LIN {X 0,Y 580.933,Z 477.254,A -85,B 0,C 180,E1 -1786.489,E2 -1786.489} C_VEL
LIN {X 0,Y 580.805,Z 577.725,A -85,B 0,C 180,E1 -1787.752,E2 -1787.752} C_VEL
LIN {X 0,Y 580.706,Z 590.474,A -85,B 0,C 180,E1 -1788.038,E2 -1788.038} C_VEL
LIN {X 0,Y 580.629,Z 603.373,A -85,B 0,C 180,E1 -1788.48,E2 -1788.48} C_VEL
LIN {X 0,Y 580.569,Z 614.719,A -85,B 0,C 180,E1 -1789.009,E2 -1789.009} C_VEL
LIN {X 0,Y 580.47,Z 626.557,A -85,B 0,C 180,E1 -1789.713,E2 -1789.713} C_VEL
LIN {X 0,Y 580.367,Z 638.111,A -85,B 0,C 180,E1 -1790.591,E2 -1790.591} C_VEL
LIN {X 0,Y 580.281,Z 647.332,A -85,B 0,C 180,E1 -1791.468,E2 -1791.468} C_VEL
LIN {X 0,Y 580.221,Z 654.959,A -85,B 0,C 180,E1 -1792.343,E2 -1792.343} C_VEL
LIN {X 0,Y 580.171,Z 662.355,A -85,B 0,C 180,E1 -1793.377,E2 -1793.377} C_VEL
LIN {X 0,Y 580.138,Z 668.453,A -85,B 0,C 180,E1 -1794.438,E2 -1794.438} C_VEL
LIN {X 0,Y 580.107,Z 673.197,A -85,B 0,C 180,E1 -1795.483,E2 -1795.483} C_VEL
LIN {X 0,Y 580.123,Z 676.829,A -85,B 0,C 180,E1 -1796.527,E2 -1796.527} C_VEL
LIN {X 0,Y 580.043,Z 678.681,A -85,B 0,C 180,E1 -1797.222,E2 -1797.222} C_VEL
LIN {X 0,Y 580.046,Z 681.138,A -85,B 0,C 180,E1 -1798.611,E2 -1798.611} C_VEL
LIN {X 0,Y 580.041,Z 681.753,A -85,B 0,C 180,E1 -1799.306,E2 -1799.306} C_VEL
LIN {X 0,Y 580.04,Z 681.812,A -85,B 0,C 180,E1 -1800.694,E2 -1800.694} C_VEL
LIN {X 0,Y 580.047,Z 681.24,A -85,B 0,C 180,E1 -1801.389,E2 -1801.389} C_VEL
LIN {X 0,Y 580.044,Z 678.908,A -85,B 0,C 180,E1 -1802.778,E2 -1802.778} C_VEL
LIN {X 0,Y 580.11,Z 676.037,A -85,B 0,C 180,E1 -1803.821,E2 -1803.821} C_VEL
LIN {X 0,Y 580.053,Z 672.134,A -85,B 0,C 180,E1 -1804.865,E2 -1804.865} C_VEL
LIN {X 0,Y 580.162,Z 667.083,A -85,B 0,C 180,E1 -1805.91,E2 -1805.91} C_VEL
LIN {X 0,Y 580.157,Z 660.739,A -85,B 0,C 180,E1 -1806.958,E2 -1806.958} C_VEL
LIN {X 0,Y 580.241,Z 652.871,A -85,B 0,C 180,E1 -1808.007,E2 -1808.007} C_VEL
LIN {X 0,Y 580.308,Z 643.003,A -85,B 0,C 180,E1 -1809.058,E2 -1809.058} C_VEL
LIN {X 0,Y 580.392,Z 633.8,A -85,B 0,C 180,E1 -1809.848,E2 -1809.848} C_VEL
LIN {X 0,Y 580.498,Z 623.854,A -85,B 0,C 180,E1 -1810.551,E2 -1810.551} C_VEL
LIN {X 0,Y 580.609,Z 613.074,A -85,B 0,C 180,E1 -1811.167,E2 -1811.167} C_VEL
LIN {X 0,Y 580.642,Z 600.005,A -85,B 0,C 180,E1 -1811.741,E2 -1811.741} C_VEL
LIN {X 0,Y 580.739,Z 587.106,A -85,B 0,C 180,E1 -1812.138,E2 -1812.138} C_VEL
LIN {X 0,Y 580.789,Z 575.132,A -85,B 0,C 180,E1 -1812.381,E2 -1812.381} C_VEL
LIN {X 0,Y 580.811,Z 472.633,A -85,B 0,C 180,E1 -1813.662,E2 -1813.662} C_VEL
LIN {X 0,Y 580.398,Z 469.615,A -85,B 0,C 180,E1 -1813.725,E2 -1813.725} C_VEL
LIN {X 0,Y 580.566,Z 448.09,A -85,B 0,C 180,E1 -1816.709,E2 -1816.709} C_VEL
LIN {X 0,Y 580.771,Z 427.235,A -85,B 0,C 180,E1 -1819.641,E2 -1819.641} C_VEL
LIN {X 0,Y 580.959,Z 406.656,A -85,B 0,C 180,E1 -1822.587,E2 -1822.587} C_VEL
LIN {X 0,Y 580.331,Z 401.637,A -85,B 0,C 180,E1 -1823.343,E2 -1823.343} C_VEL
LIN {X 0,Y 580.262,Z 401.208,A -85,B 0,C 180,E1 -1823.417,E2 -1823.417} C_VEL
LIN {X 0,Y 580.26,Z 401.203,A -85,B 0,C 180,E1 -1826.327,E2 -1826.327} C_VEL
LIN {X 0,Y 580.278,Z 401.204,A -85,B 0,C 180,E1 -1829.305,E2 -1829.305} C_VEL
LIN {X 0,Y 580.296,Z 401.197,A -85,B 0,C 180,E1 -1832.201,E2 -1832.201} C_VEL
LIN {X 0,Y 580.288,Z 401.198,A -85,B 0,C 180,E1 -1834.697,E2 -1834.697} C_VEL
LIN {X 0,Y 580.291,Z 401.205,A -85,B 0,C 180,E1 -1837.269,E2 -1837.269} C_VEL
LIN {X 0,Y 580.293,Z 401.196,A -85,B 0,C 180,E1 -1840.27,E2 -1840.27} C_VEL
LIN {X 0,Y 580.28,Z 401.202,A -85,B 0,C 180,E1 -1842.706,E2 -1842.706} C_VEL
LIN {X 0,Y 580.274,Z 401.2,A -85,B 0,C 180,E1 -1845.609,E2 -1845.609} C_VEL
LIN {X 0,Y 580.284,Z 401.199,A -85,B 0,C 180,E1 -1848.231,E2 -1848.231} C_VEL
LIN {X 0,Y 580.277,Z 401.205,A -85,B 0,C 180,E1 -1850.965,E2 -1850.965} C_VEL
LIN {X 0,Y 580.251,Z 401.201,A -85,B 0,C 180,E1 -1853.595,E2 -1853.595} C_VEL
LIN {X 0,Y 580.315,Z 401.197,A -85,B 0,C 180,E1 -1856.145,E2 -1856.145} C_VEL
LIN {X 0,Y 580.269,Z 401.207,A -85,B 0,C 180,E1 -1858.614,E2 -1858.614} C_VEL
LIN {X 0,Y 580.285,Z 401.2,A -85,B 0,C 180,E1 -1861.023,E2 -1861.023} C_VEL
LIN {X 0,Y 580.301,Z 401.201,A -85,B 0,C 180,E1 -1864.344,E2 -1864.344} C_VEL
LIN {X 0,Y 581.342,Z 407.343,A -85,B 0,C 180,E1 -1865.202,E2 -1865.202} C_VEL
LIN {X 0,Y 581.077,Z 429.583,A -85,B 0,C 180,E1 -1867.979,E2 -1867.979} C_VEL
LIN {X 0,Y 580.889,Z 450.217,A -85,B 0,C 180,E1 -1870.512,E2 -1870.512} C_VEL
LIN {X 0,Y 580.646,Z 473.238,A -85,B 0,C 180,E1 -1873.294,E2 -1873.294} C_VEL
LIN {X 0,Y 580.433,Z 498.075,A -85,B 0,C 180,E1 -1876.254,E2 -1876.254} C_VEL
LIN {X 0,Y 580.423,Z 498.64,A -85,B 0,C 180,E1 -1876.32,E2 -1876.32} C_VEL
LIN {X 0,Y 580.919,Z 503.714,A -85,B 0,C 180,E1 -1876.399,E2 -1876.399} C_VEL
LIN {X 0,Y 580.797,Z 607.943,A -85,B 0,C 180,E1 -1877.708,E2 -1877.708} C_VEL
LIN {X 0,Y 580.735,Z 621.217,A -85,B 0,C 180,E1 -1878.017,E2 -1878.017} C_VEL
LIN {X 0,Y 580.644,Z 634.148,A -85,B 0,C 180,E1 -1878.467,E2 -1878.467} C_VEL
LIN {X 0,Y 580.556,Z 645.629,A -85,B 0,C 180,E1 -1879.008,E2 -1879.008} C_VEL
LIN {X 0,Y 580.428,Z 657.202,A -85,B 0,C 180,E1 -1879.712,E2 -1879.712} C_VEL
LIN {X 0,Y 580.344,Z 667.598,A -85,B 0,C 180,E1 -1880.503,E2 -1880.503} C_VEL
LIN {X 0,Y 580.271,Z 676.112,A -85,B 0,C 180,E1 -1881.292,E2 -1881.292} C_VEL
LIN {X 0,Y 580.222,Z 683.96,A -85,B 0,C 180,E1 -1882.168,E2 -1882.168} C_VEL
LIN {X 0,Y 580.154,Z 691.65,A -85,B 0,C 180,E1 -1883.222,E2 -1883.222} C_VEL
LIN {X 0,Y 580.139,Z 698.68,A -85,B 0,C 180,E1 -1884.438,E2 -1884.438} C_VEL
LIN {X 0,Y 580.108,Z 703.372,A -85,B 0,C 180,E1 -1885.483,E2 -1885.483} C_VEL
LIN {X 0,Y 580.123,Z 706.957,A -85,B 0,C 180,E1 -1886.527,E2 -1886.527} C_VEL
LIN {X 0,Y 580.043,Z 708.808,A -85,B 0,C 180,E1 -1887.222,E2 -1887.222} C_VEL
LIN {X 0,Y 580.039,Z 710.199,A -85,B 0,C 180,E1 -1887.917,E2 -1887.917} C_VEL
LIN {X 0,Y 580.04,Z 711.785,A -85,B 0,C 180,E1 -1889.306,E2 -1889.306} C_VEL
LIN {X 0,Y 580.037,Z 712,A -85,B 0,C 180,E1 -1890,E2 -1890} C_VEL
LIN {X 0,Y 580.046,Z 711.186,A -85,B 0,C 180,E1 -1891.389,E2 -1891.389} C_VEL
LIN {X 0,Y 580.039,Z 710.2,A -85,B 0,C 180,E1 -1892.083,E2 -1892.083} C_VEL
LIN {X 0,Y 580.043,Z 708.81,A -85,B 0,C 180,E1 -1892.778,E2 -1892.778} C_VEL
LIN {X 0,Y 580.11,Z 705.896,A -85,B 0,C 180,E1 -1893.821,E2 -1893.821} C_VEL
LIN {X 0,Y 580.053,Z 701.949,A -85,B 0,C 180,E1 -1894.865,E2 -1894.865} C_VEL
LIN {X 0,Y 580.139,Z 695.877,A -85,B 0,C 180,E1 -1896.085,E2 -1896.085} C_VEL
LIN {X 0,Y 580.184,Z 689.237,A -85,B 0,C 180,E1 -1897.132,E2 -1897.132} C_VEL
LIN {X 0,Y 580.251,Z 680.99,A -85,B 0,C 180,E1 -1898.182,E2 -1898.182} C_VEL
LIN {X 0,Y 580.308,Z 672.537,A -85,B 0,C 180,E1 -1899.058,E2 -1899.058} C_VEL
LIN {X 0,Y 580.419,Z 662.096,A -85,B 0,C 180,E1 -1899.936,E2 -1899.936} C_VEL
LIN {X 0,Y 580.512,Z 651.756,A -85,B 0,C 180,E1 -1900.639,E2 -1900.639} C_VEL
LIN {X 0,Y 580.581,Z 640.408,A -85,B 0,C 180,E1 -1901.256,E2 -1901.256} C_VEL
LIN {X 0,Y 580.65,Z 628.765,A -85,B 0,C 180,E1 -1901.741,E2 -1901.741} C_VEL
LIN {X 0,Y 580.748,Z 615.347,A -85,B 0,C 180,E1 -1902.138,E2 -1902.138} C_VEL
LIN {X 0,Y 580.817,Z 602.079,A -85,B 0,C 180,E1 -1902.38,E2 -1902.38} C_VEL
LIN {X 0,Y 580.879,Z 501.925,A -85,B 0,C 180,E1 -1903.624,E2 -1903.624} C_VEL
LIN {X 0,Y 580.424,Z 498.452,A -85,B 0,C 180,E1 -1903.702,E2 -1903.702} C_VEL
LIN {X 0,Y 580.636,Z 474.743,A -85,B 0,C 180,E1 -1906.526,E2 -1906.526} C_VEL
LIN {X 0,Y 580.87,Z 451.661,A -85,B 0,C 180,E1 -1909.312,E2 -1909.312} C_VEL
LIN {X 0,Y 581.077,Z 429.583,A -85,B 0,C 180,E1 -1912.021,E2 -1912.021} C_VEL
LIN {X 0,Y 581.331,Z 407.325,A -85,B 0,C 180,E1 -1914.801,E2 -1914.801} C_VEL
LIN {X 0,Y 580.288,Z 401.206,A -85,B 0,C 180,E1 -1915.633,E2 -1915.633} C_VEL
LIN {X 0,Y 580.248,Z 401.205,A -85,B 0,C 180,E1 -1918.188,E2 -1918.188} C_VEL
LIN {X 0,Y 580.271,Z 401.2,A -85,B 0,C 180,E1 -1920.692,E2 -1920.692} C_VEL
LIN {X 0,Y 580.304,Z 401.201,A -85,B 0,C 180,E1 -1923.316,E2 -1923.316} C_VEL
LIN {X 0,Y 580.234,Z 401.209,A -85,B 0,C 180,E1 -1925.754,E2 -1925.754} C_VEL
LIN {X 0,Y 580.286,Z 401.198,A -85,B 0,C 180,E1 -1928.147,E2 -1928.147} C_VEL
LIN {X 0,Y 580.298,Z 401.198,A -85,B 0,C 180,E1 -1930.844,E2 -1930.844} C_VEL
LIN {X 0,Y 580.273,Z 401.203,A -85,B 0,C 180,E1 -1933.659,E2 -1933.659} C_VEL
LIN {X 0,Y 580.279,Z 401.199,A -85,B 0,C 180,E1 -1936.61,E2 -1936.61} C_VEL
LIN {X 0,Y 580.3,Z 401.205,A -85,B 0,C 180,E1 -1939.157,E2 -1939.157} C_VEL
LIN {X 0,Y 580.293,Z 401.196,A -85,B 0,C 180,E1 -1941.927,E2 -1941.927} C_VEL
LIN {X 0,Y 580.255,Z 401.203,A -85,B 0,C 180,E1 -1944.453,E2 -1944.453} C_VEL
LIN {X 0,Y 580.291,Z 401.205,A -85,B 0,C 180,E1 -1946.975,E2 -1946.975} C_VEL
LIN {X 0,Y 580.299,Z 401.198,A -85,B 0,C 180,E1 -1949.425,E2 -1949.425} C_VEL
LIN {X 0,Y 580.299,Z 401.197,A -85,B 0,C 180,E1 -1952.142,E2 -1952.142} C_VEL
LIN {X 0,Y 580.324,Z 401.195,A -85,B 0,C 180,E1 -1955.27,E2 -1955.27} C_VEL
LIN {X 0,Y 580.271,Z 401.2,A -85,B 0,C 180,E1 -1957.947,E2 -1957.947} C_VEL
LIN {X 0,Y 580.288,Z 401.202,A -85,B 0,C 180,E1 -1960.913,E2 -1960.913} C_VEL
LIN {X 0,Y 580.289,Z 401.199,A -85,B 0,C 180,E1 -1963.102,E2 -1963.102} C_VEL
LIN {X 0,Y 580.281,Z 401.203,A -85,B 0,C 180,E1 -1965.982,E2 -1965.982} C_VEL
LIN {X 0,Y 580.25,Z 402.922,A -85,B 0,C 180,E1 -1966.417,E2 -1966.417} C_VEL
LIN {X 0,Y 580.983,Z 409.047,A -85,B 0,C 180,E1 -1966.512,E2 -1966.512} C_VEL
LIN {X 0,Y 580.789,Z 507.728,A -85,B 0,C 180,E1 -1967.752,E2 -1967.752} C_VEL
LIN {X 0,Y 580.725,Z 521.239,A -85,B 0,C 180,E1 -1968.061,E2 -1968.061} C_VEL
LIN {X 0,Y 580.665,Z 533.35,A -85,B 0,C 180,E1 -1968.481,E2 -1968.481} C_VEL
LIN {X 0,Y 580.555,Z 544.709,A -85,B 0,C 180,E1 -1969.008,E2 -1969.008} C_VEL
LIN {X 0,Y 580.456,Z 555.204,A -85,B 0,C 180,E1 -1969.624,E2 -1969.624} C_VEL
LIN {X 0,Y 580.361,Z 566.006,A -85,B 0,C 180,E1 -1970.415,E2 -1970.415} C_VEL
LIN {X 0,Y 580.272,Z 575.649,A -85,B 0,C 180,E1 -1971.292,E2 -1971.292} C_VEL
LIN {X 0,Y 580.222,Z 583.547,A -85,B 0,C 180,E1 -1972.168,E2 -1972.168} C_VEL
LIN {X 0,Y 580.168,Z 591.284,A -85,B 0,C 180,E1 -1973.21,E2 -1973.21} C_VEL
LIN {X 0,Y 580.139,Z 598.456,A -85,B 0,C 180,E1 -1974.438,E2 -1974.438} C_VEL
LIN {X 0,Y 580.108,Z 603.188,A -85,B 0,C 180,E1 -1975.483,E2 -1975.483} C_VEL
LIN {X 0,Y 580.123,Z 606.809,A -85,B 0,C 180,E1 -1976.527,E2 -1976.527} C_VEL
LIN {X 0,Y 580.043,Z 608.701,A -85,B 0,C 180,E1 -1977.222,E2 -1977.222} C_VEL
LIN {X 0,Y 580.039,Z 610.133,A -85,B 0,C 180,E1 -1977.917,E2 -1977.917} C_VEL
LIN {X 0,Y 580.04,Z 611.759,A -85,B 0,C 180,E1 -1979.306,E2 -1979.306} C_VEL
LIN {X 0,Y 580.038,Z 611.996,A -85,B 0,C 180,E1 -1980,E2 -1980} C_VEL
LIN {X 0,Y 580.047,Z 611.227,A -85,B 0,C 180,E1 -1981.389,E2 -1981.389} C_VEL
LIN {X 0,Y 580.04,Z 610.28,A -85,B 0,C 180,E1 -1982.083,E2 -1982.083} C_VEL
LIN {X 0,Y 580.044,Z 608.892,A -85,B 0,C 180,E1 -1982.778,E2 -1982.778} C_VEL
LIN {X 0,Y 580.11,Z 606.026,A -85,B 0,C 180,E1 -1983.821,E2 -1983.821} C_VEL
LIN {X 0,Y 580.054,Z 602.136,A -85,B 0,C 180,E1 -1984.865,E2 -1984.865} C_VEL
LIN {X 0,Y 580.141,Z 596.116,A -85,B 0,C 180,E1 -1986.085,E2 -1986.085} C_VEL
LIN {X 0,Y 580.185,Z 589.531,A -85,B 0,C 180,E1 -1987.132,E2 -1987.132} C_VEL
LIN {X 0,Y 580.246,Z 581.368,A -85,B 0,C 180,E1 -1988.182,E2 -1988.182} C_VEL
LIN {X 0,Y 580.308,Z 573.014,A -85,B 0,C 180,E1 -1989.058,E2 -1989.058} C_VEL
LIN {X 0,Y 580.419,Z 562.657,A -85,B 0,C 180,E1 -1989.936,E2 -1989.936} C_VEL
LIN {X 0,Y 580.494,Z 552.438,A -85,B 0,C 180,E1 -1990.64,E2 -1990.64} C_VEL
LIN {X 0,Y 580.612,Z 541.308,A -85,B 0,C 180,E1 -1991.255,E2 -1991.255} C_VEL
LIN {X 0,Y 580.651,Z 528.748,A -85,B 0,C 180,E1 -1991.786,E2 -1991.786} C_VEL
LIN {X 0,Y 580.754,Z 516.199,A -85,B 0,C 180,E1 -1992.16,E2 -1992.16} C_VEL
LIN {X 0,Y 580.84,Z 503.638,A -85,B 0,C 180,E1 -1992.402,E2 -1992.402} C_VEL
LIN {X 0,Y 580.905,Z 458.36,A -85,B 0,C 180,E1 -1992.966,E2 -1992.966} C_VEL
LIN {X 0,Y 580.247,Z 452.555,A -85,B 0,C 180,E1 -1993.053,E2 -1993.053} C_VEL
LIN {X 0,Y 574.723,Z 433.865,A -85,B 0,C 180,E1 -1993.416,E2 -1993.416} C_VEL
LIN {X 0,Y 574.066,Z 428.061,A -85,B 0,C 180,E1 -1993.504,E2 -1993.504} C_VEL
LIN {X 0,Y 573.912,Z 407.178,A -85,B 0,C 180,E1 -1993.771,E2 -1993.771} C_VEL
LIN {X 0,Y 573.186,Z 402.872,A -85,B 0,C 180,E1 -1993.856,E2 -1993.856} C_VEL
LIN {X 0,Y 573.186,Z 402.087,A -85,B 0,C 180,E1 -1994.059,E2 -1994.059} C_VEL
LIN {X 0,Y 573.22,Z 402.08,A -85,B 0,C 180,E1 -1996.995,E2 -1996.995} C_VEL
LIN {X 0,Y 573.239,Z 402.077,A -85,B 0,C 180,E1 -2000.077,E2 -2000.077} C_VEL
LIN {X 0,Y 573.227,Z 402.076,A -85,B 0,C 180,E1 -2002.338,E2 -2002.338} C_VEL
LIN {X 0,Y 573.237,Z 402.083,A -85,B 0,C 180,E1 -2005.411,E2 -2005.411} C_VEL
LIN {X 0,Y 573.234,Z 402.075,A -85,B 0,C 180,E1 -2008.565,E2 -2008.565} C_VEL
LIN {X 0,Y 573.229,Z 402.083,A -85,B 0,C 180,E1 -2010.993,E2 -2010.993} C_VEL
LIN {X 0,Y 573.266,Z 402.072,A -85,B 0,C 180,E1 -2013.524,E2 -2013.524} C_VEL
LIN {X 0,Y 573.218,Z 402.077,A -85,B 0,C 180,E1 -2016.052,E2 -2016.052} C_VEL
LIN {X 0,Y 573.246,Z 402.079,A -85,B 0,C 180,E1 -2018.701,E2 -2018.701} C_VEL
LIN {X 0,Y 573.234,Z 402.076,A -85,B 0,C 180,E1 -2021.593,E2 -2021.593} C_VEL
LIN {X 0,Y 573.237,Z 402.078,A -85,B 0,C 180,E1 -2024.334,E2 -2024.334} C_VEL
LIN {X 0,Y 573.246,Z 402.075,A -85,B 0,C 180,E1 -2027.358,E2 -2027.358} C_VEL
LIN {X 0,Y 573.24,Z 402.079,A -85,B 0,C 180,E1 -2030.392,E2 -2030.392} C_VEL
LIN {X 0,Y 573.233,Z 402.078,A -85,B 0,C 180,E1 -2033.076,E2 -2033.076} C_VEL
LIN {X 0,Y 573.265,Z 402.071,A -85,B 0,C 180,E1 -2035.671,E2 -2035.671} C_VEL
LIN {X 0,Y 573.238,Z 402.081,A -85,B 0,C 180,E1 -2038.184,E2 -2038.184} C_VEL
LIN {X 0,Y 573.243,Z 402.081,A -85,B 0,C 180,E1 -2040.633,E2 -2040.633} C_VEL
LIN {X 0,Y 573.204,Z 402.081,A -85,B 0,C 180,E1 -2043.515,E2 -2043.515} C_VEL
LIN {X 0,Y 573.218,Z 402.087,A -85,B 0,C 180,E1 -2046.417,E2 -2046.417} C_VEL
LIN {X 0,Y 573.244,Z 402.244,A -85,B 0,C 180,E1 -2046.535,E2 -2046.535} C_VEL
LIN {X 0,Y 574.049,Z 407.333,A -85,B 0,C 180,E1 -2047.316,E2 -2047.316} C_VEL
LIN {X 0,Y 573.81,Z 428.297,A -85,B 0,C 180,E1 -2050.354,E2 -2050.354} C_VEL
LIN {X 0,Y 573.567,Z 448.837,A -85,B 0,C 180,E1 -2053.278,E2 -2053.278} C_VEL
LIN {X 0,Y 573.392,Z 469.614,A -85,B 0,C 180,E1 -2056.194,E2 -2056.194} C_VEL
LIN {X 0,Y 574.037,Z 475.513,A -85,B 0,C 180,E1 -2056.301,E2 -2056.301} C_VEL
LIN {X 0,Y 573.869,Z 577.679,A -85,B 0,C 180,E1 -2057.602,E2 -2057.602} C_VEL
LIN {X 0,Y 573.792,Z 589.623,A -85,B 0,C 180,E1 -2057.87,E2 -2057.87} C_VEL
LIN {X 0,Y 573.697,Z 603.399,A -85,B 0,C 180,E1 -2058.339,E2 -2058.339} C_VEL
LIN {X 0,Y 573.582,Z 614.865,A -85,B 0,C 180,E1 -2058.879,E2 -2058.879} C_VEL
LIN {X 0,Y 573.48,Z 625.186,A -85,B 0,C 180,E1 -2059.497,E2 -2059.497} C_VEL
LIN {X 0,Y 573.361,Z 634.874,A -85,B 0,C 180,E1 -2060.208,E2 -2060.208} C_VEL
LIN {X 0,Y 573.277,Z 643.853,A -85,B 0,C 180,E1 -2061.007,E2 -2061.007} C_VEL
LIN {X 0,Y 573.178,Z 652.102,A -85,B 0,C 180,E1 -2061.894,E2 -2061.894} C_VEL
LIN {X 0,Y 573.105,Z 660.164,A -85,B 0,C 180,E1 -2062.956,E2 -2062.956} C_VEL
LIN {X 0,Y 573.094,Z 666.617,A -85,B 0,C 180,E1 -2064.017,E2 -2064.017} C_VEL
LIN {X 0,Y 572.962,Z 671.738,A -85,B 0,C 180,E1 -2065.074,E2 -2065.074} C_VEL
LIN {X 0,Y 573.014,Z 675.723,A -85,B 0,C 180,E1 -2066.132,E2 -2066.132} C_VEL
LIN {X 0,Y 572.959,Z 678.679,A -85,B 0,C 180,E1 -2067.188,E2 -2067.188} C_VEL
LIN {X 0,Y 572.939,Z 680.137,A -85,B 0,C 180,E1 -2067.891,E2 -2067.891} C_VEL
LIN {X 0,Y 572.941,Z 681.753,A -85,B 0,C 180,E1 -2069.297,E2 -2069.297} C_VEL
LIN {X 0,Y 572.939,Z 681.996,A -85,B 0,C 180,E1 -2070,E2 -2070} C_VEL
LIN {X 0,Y 572.947,Z 681.231,A -85,B 0,C 180,E1 -2071.406,E2 -2071.406} C_VEL
LIN {X 0,Y 572.939,Z 680.278,A -85,B 0,C 180,E1 -2072.109,E2 -2072.109} C_VEL
LIN {X 0,Y 573.022,Z 677.072,A -85,B 0,C 180,E1 -2073.516,E2 -2073.516} C_VEL
LIN {X 0,Y 573.029,Z 673.52,A -85,B 0,C 180,E1 -2074.573,E2 -2074.573} C_VEL
LIN {X 0,Y 573.068,Z 668.874,A -85,B 0,C 180,E1 -2075.63,E2 -2075.63} C_VEL
LIN {X 0,Y 573.07,Z 662.933,A -85,B 0,C 180,E1 -2076.7,E2 -2076.7} C_VEL
LIN {X 0,Y 573.16,Z 655.675,A -85,B 0,C 180,E1 -2077.752,E2 -2077.752} C_VEL
LIN {X 0,Y 573.232,Z 646.556,A -85,B 0,C 180,E1 -2078.816,E2 -2078.816} C_VEL
LIN {X 0,Y 573.337,Z 637.061,A -85,B 0,C 180,E1 -2079.703,E2 -2079.703} C_VEL
LIN {X 0,Y 573.434,Z 627.817,A -85,B 0,C 180,E1 -2080.415,E2 -2080.415} C_VEL
LIN {X 0,Y 573.554,Z 617.963,A -85,B 0,C 180,E1 -2081.037,E2 -2081.037} C_VEL
LIN {X 0,Y 573.645,Z 606.66,A -85,B 0,C 180,E1 -2081.608,E2 -2081.608} C_VEL
LIN {X 0,Y 573.765,Z 594.827,A -85,B 0,C 180,E1 -2082.064,E2 -2082.064} C_VEL
LIN {X 0,Y 573.822,Z 581.405,A -85,B 0,C 180,E1 -2082.421,E2 -2082.421} C_VEL
LIN {X 0,Y 573.914,Z 563.154,A -85,B 0,C 180,E1 -2082.689,E2 -2082.689} C_VEL
LIN {X 0,Y 573.962,Z 473.702,A -85,B 0,C 180,E1 -2083.814,E2 -2083.814} C_VEL
LIN {X 0,Y 573.409,Z 469.611,A -85,B 0,C 180,E1 -2083.896,E2 -2083.896} C_VEL
LIN {X 0,Y 573.569,Z 449.469,A -85,B 0,C 180,E1 -2086.723,E2 -2086.723} C_VEL
LIN {X 0,Y 573.816,Z 428.666,A -85,B 0,C 180,E1 -2089.683,E2 -2089.683} C_VEL
LIN {X 0,Y 574.041,Z 407.946,A -85,B 0,C 180,E1 -2092.685,E2 -2092.685} C_VEL
LIN {X 0,Y 573.647,Z 404.285,A -85,B 0,C 180,E1 -2093.24,E2 -2093.24} C_VEL
LIN {X 0,Y 573.22,Z 402.086,A -85,B 0,C 180,E1 -2093.593,E2 -2093.593} C_VEL
LIN {X 0,Y 573.202,Z 402.082,A -85,B 0,C 180,E1 -2096.485,E2 -2096.485} C_VEL
LIN {X 0,Y 573.243,Z 402.08,A -85,B 0,C 180,E1 -2099.367,E2 -2099.367} C_VEL
LIN {X 0,Y 573.25,Z 402.075,A -85,B 0,C 180,E1 -2102.227,E2 -2102.227} C_VEL
LIN {X 0,Y 573.234,Z 402.077,A -85,B 0,C 180,E1 -2104.771,E2 -2104.771} C_VEL
LIN {X 0,Y 573.233,Z 402.078,A -85,B 0,C 180,E1 -2107.808,E2 -2107.808} C_VEL
LIN {X 0,Y 573.248,Z 402.074,A -85,B 0,C 180,E1 -2110.525,E2 -2110.525} C_VEL
LIN {X 0,Y 573.242,Z 402.079,A -85,B 0,C 180,E1 -2113.359,E2 -2113.359} C_VEL
LIN {X 0,Y 573.248,Z 402.075,A -85,B 0,C 180,E1 -2116.331,E2 -2116.331} C_VEL
LIN {X 0,Y 573.233,Z 402.078,A -85,B 0,C 180,E1 -2118.543,E2 -2118.543} C_VEL
LIN {X 0,Y 573.248,Z 402.076,A -85,B 0,C 180,E1 -2121.299,E2 -2121.299} C_VEL
LIN {X 0,Y 573.196,Z 402.079,A -85,B 0,C 180,E1 -2124.021,E2 -2124.021} C_VEL
LIN {X 0,Y 573.273,Z 402.078,A -85,B 0,C 180,E1 -2126.518,E2 -2126.518} C_VEL
LIN {X 0,Y 573.224,Z 402.079,A -85,B 0,C 180,E1 -2129.119,E2 -2129.119} C_VEL
LIN {X 0,Y 573.209,Z 402.079,A -85,B 0,C 180,E1 -2131.434,E2 -2131.434} C_VEL
LIN {X 0,Y 573.234,Z 402.083,A -85,B 0,C 180,E1 -2134.589,E2 -2134.589} C_VEL
LIN {X 0,Y 573.245,Z 402.249,A -85,B 0,C 180,E1 -2136.535,E2 -2136.535} C_VEL
LIN {X 0,Y 574.017,Z 407.333,A -85,B 0,C 180,E1 -2137.314,E2 -2137.314} C_VEL
LIN {X 0,Y 573.832,Z 426.745,A -85,B 0,C 180,E1 -2140.131,E2 -2140.131} C_VEL
LIN {X 0,Y 573.589,Z 446.979,A -85,B 0,C 180,E1 -2143.015,E2 -2143.015} C_VEL
LIN {X 0,Y 573.421,Z 468.158,A -85,B 0,C 180,E1 -2145.992,E2 -2145.992} C_VEL
LIN {X 0,Y 573.392,Z 469.614,A -85,B 0,C 180,E1 -2146.194,E2 -2146.194} C_VEL
LIN {X 0,Y 574.037,Z 475.511,A -85,B 0,C 180,E1 -2146.301,E2 -2146.301} C_VEL
LIN {X 0,Y 573.869,Z 577.711,A -85,B 0,C 180,E1 -2147.602,E2 -2147.602} C_VEL
LIN {X 0,Y 573.779,Z 590.502,A -85,B 0,C 180,E1 -2147.892,E2 -2147.892} C_VEL
LIN {X 0,Y 573.663,Z 603.381,A -85,B 0,C 180,E1 -2148.338,E2 -2148.338} C_VEL
LIN {X 0,Y 573.594,Z 615.003,A -85,B 0,C 180,E1 -2148.889,E2 -2148.889} C_VEL
LIN {X 0,Y 573.466,Z 625.19,A -85,B 0,C 180,E1 -2149.496,E2 -2149.496} C_VEL
LIN {X 0,Y 573.348,Z 636.018,A -85,B 0,C 180,E1 -2150.297,E2 -2150.297} C_VEL
LIN {X 0,Y 573.241,Z 645.668,A -85,B 0,C 180,E1 -2151.185,E2 -2151.185} C_VEL
LIN {X 0,Y 573.161,Z 653.556,A -85,B 0,C 180,E1 -2152.071,E2 -2152.071} C_VEL
LIN {X 0,Y 573.112,Z 660.13,A -85,B 0,C 180,E1 -2152.956,E2 -2152.956} C_VEL
LIN {X 0,Y 573.076,Z 666.579,A -85,B 0,C 180,E1 -2154.017,E2 -2154.017} C_VEL
LIN {X 0,Y 572.962,Z 671.726,A -85,B 0,C 180,E1 -2155.074,E2 -2155.074} C_VEL
LIN {X 0,Y 573.014,Z 675.721,A -85,B 0,C 180,E1 -2156.132,E2 -2156.132} C_VEL
LIN {X 0,Y 572.959,Z 678.679,A -85,B 0,C 180,E1 -2157.188,E2 -2157.188} C_VEL
LIN {X 0,Y 572.946,Z 681.14,A -85,B 0,C 180,E1 -2158.594,E2 -2158.594} C_VEL
LIN {X 0,Y 572.941,Z 681.753,A -85,B 0,C 180,E1 -2159.297,E2 -2159.297} C_VEL
LIN {X 0,Y 572.94,Z 681.811,A -85,B 0,C 180,E1 -2160.703,E2 -2160.703} C_VEL
LIN {X 0,Y 572.947,Z 681.241,A -85,B 0,C 180,E1 -2161.406,E2 -2161.406} C_VEL
LIN {X 0,Y 572.96,Z 678.904,A -85,B 0,C 180,E1 -2162.812,E2 -2162.812} C_VEL
LIN {X 0,Y 573.015,Z 676.031,A -85,B 0,C 180,E1 -2163.868,E2 -2163.868} C_VEL
LIN {X 0,Y 572.963,Z 672.124,A -85,B 0,C 180,E1 -2164.926,E2 -2164.926} C_VEL
LIN {X 0,Y 573.076,Z 667.071,A -85,B 0,C 180,E1 -2165.983,E2 -2165.983} C_VEL
LIN {X 0,Y 573.082,Z 660.726,A -85,B 0,C 180,E1 -2167.044,E2 -2167.044} C_VEL
LIN {X 0,Y 573.175,Z 652.866,A -85,B 0,C 180,E1 -2168.106,E2 -2168.106} C_VEL
LIN {X 0,Y 573.287,Z 642.991,A -85,B 0,C 180,E1 -2169.17,E2 -2169.17} C_VEL
LIN {X 0,Y 573.397,Z 633.783,A -85,B 0,C 180,E1 -2169.97,E2 -2169.97} C_VEL
LIN {X 0,Y 573.507,Z 623.844,A -85,B 0,C 180,E1 -2170.681,E2 -2170.681} C_VEL
LIN {X 0,Y 573.629,Z 613.065,A -85,B 0,C 180,E1 -2171.305,E2 -2171.305} C_VEL
LIN {X 0,Y 573.676,Z 599.978,A -85,B 0,C 180,E1 -2171.886,E2 -2171.886} C_VEL
LIN {X 0,Y 573.811,Z 587.936,A -85,B 0,C 180,E1 -2172.265,E2 -2172.265} C_VEL
LIN {X 0,Y 573.881,Z 576.388,A -85,B 0,C 180,E1 -2172.51,E2 -2172.51} C_VEL
LIN {X 0,Y 573.962,Z 473.705,A -85,B 0,C 180,E1 -2173.814,E2 -2173.814} C_VEL
LIN {X 0,Y 573.407,Z 469.611,A -85,B 0,C 180,E1 -2173.896,E2 -2173.896} C_VEL
LIN {X 0,Y 573.568,Z 449.47,A -85,B 0,C 180,E1 -2176.723,E2 -2176.723} C_VEL
LIN {X 0,Y 573.81,Z 428.923,A -85,B 0,C 180,E1 -2179.646,E2 -2179.646} C_VEL
LIN {X 0,Y 574.059,Z 409.241,A -85,B 0,C 180,E1 -2182.494,E2 -2182.494} C_VEL
LIN {X 0,Y 573.652,Z 404.275,A -85,B 0,C 180,E1 -2183.241,E2 -2183.241} C_VEL
LIN {X 0,Y 573.22,Z 402.086,A -85,B 0,C 180,E1 -2183.593,E2 -2183.593} C_VEL
LIN {X 0,Y 573.202,Z 402.081,A -85,B 0,C 180,E1 -2186.485,E2 -2186.485} C_VEL
LIN {X 0,Y 573.243,Z 402.081,A -85,B 0,C 180,E1 -2189.367,E2 -2189.367} C_VEL
LIN {X 0,Y 573.25,Z 402.075,A -85,B 0,C 180,E1 -2192.227,E2 -2192.227} C_VEL
LIN {X 0,Y 573.234,Z 402.077,A -85,B 0,C 180,E1 -2194.771,E2 -2194.771} C_VEL
LIN {X 0,Y 573.233,Z 402.078,A -85,B 0,C 180,E1 -2197.808,E2 -2197.808} C_VEL
LIN {X 0,Y 573.248,Z 402.075,A -85,B 0,C 180,E1 -2200.525,E2 -2200.525} C_VEL
LIN {X 0,Y 573.242,Z 402.08,A -85,B 0,C 180,E1 -2203.359,E2 -2203.359} C_VEL
LIN {X 0,Y 573.247,Z 402.076,A -85,B 0,C 180,E1 -2206.331,E2 -2206.331} C_VEL
LIN {X 0,Y 573.233,Z 402.08,A -85,B 0,C 180,E1 -2208.543,E2 -2208.543} C_VEL
LIN {X 0,Y 573.242,Z 402.077,A -85,B 0,C 180,E1 -2211.298,E2 -2211.298} C_VEL
LIN {X 0,Y 573.196,Z 402.082,A -85,B 0,C 180,E1 -2214.021,E2 -2214.021} C_VEL
LIN {X 0,Y 573.272,Z 402.079,A -85,B 0,C 180,E1 -2216.518,E2 -2216.518} C_VEL
LIN {X 0,Y 573.223,Z 402.079,A -85,B 0,C 180,E1 -2219.119,E2 -2219.119} C_VEL
LIN {X 0,Y 573.208,Z 402.08,A -85,B 0,C 180,E1 -2221.434,E2 -2221.434} C_VEL
LIN {X 0,Y 573.271,Z 402.158,A -85,B 0,C 180,E1 -2224.226,E2 -2224.226} C_VEL
LIN {X 0,Y 574.501,Z 409.324,A -85,B 0,C 180,E1 -2225.164,E2 -2225.164} C_VEL
LIN {X 0,Y 574.204,Z 431.089,A -85,B 0,C 180,E1 -2227.891,E2 -2227.891} C_VEL
LIN {X 0,Y 573.939,Z 452.44,A -85,B 0,C 180,E1 -2230.542,E2 -2230.542} C_VEL
LIN {X 0,Y 573.691,Z 477.754,A -85,B 0,C 180,E1 -2233.635,E2 -2233.635} C_VEL
LIN {X 0,Y 573.434,Z 498.64,A -85,B 0,C 180,E1 -2236.15,E2 -2236.15} C_VEL
LIN {X 0,Y 574.021,Z 503.714,A -85,B 0,C 180,E1 -2236.232,E2 -2236.232} C_VEL
LIN {X 0,Y 573.884,Z 607.943,A -85,B 0,C 180,E1 -2237.557,E2 -2237.557} C_VEL
LIN {X 0,Y 573.794,Z 621.217,A -85,B 0,C 180,E1 -2237.87,E2 -2237.87} C_VEL
LIN {X 0,Y 573.692,Z 634.15,A -85,B 0,C 180,E1 -2238.325,E2 -2238.325} C_VEL
LIN {X 0,Y 573.591,Z 645.632,A -85,B 0,C 180,E1 -2238.873,E2 -2238.873} C_VEL
LIN {X 0,Y 573.44,Z 657.201,A -85,B 0,C 180,E1 -2239.585,E2 -2239.585} C_VEL
LIN {X 0,Y 573.331,Z 667.599,A -85,B 0,C 180,E1 -2240.385,E2 -2240.385} C_VEL
LIN {X 0,Y 573.241,Z 676.112,A -85,B 0,C 180,E1 -2241.185,E2 -2241.185} C_VEL
LIN {X 0,Y 573.161,Z 683.96,A -85,B 0,C 180,E1 -2242.071,E2 -2242.071} C_VEL
LIN {X 0,Y 573.073,Z 691.954,A -85,B 0,C 180,E1 -2243.185,E2 -2243.185} C_VEL
LIN {X 0,Y 573.07,Z 698.68,A -85,B 0,C 180,E1 -2244.37,E2 -2244.37} C_VEL
LIN {X 0,Y 573.028,Z 703.372,A -85,B 0,C 180,E1 -2245.427,E2 -2245.427} C_VEL
LIN {X 0,Y 573.022,Z 706.957,A -85,B 0,C 180,E1 -2246.484,E2 -2246.484} C_VEL
LIN {X 0,Y 572.959,Z 708.808,A -85,B 0,C 180,E1 -2247.188,E2 -2247.188} C_VEL
LIN {X 0,Y 572.939,Z 710.198,A -85,B 0,C 180,E1 -2247.891,E2 -2247.891} C_VEL
LIN {X 0,Y 572.94,Z 711.785,A -85,B 0,C 180,E1 -2249.297,E2 -2249.297} C_VEL
LIN {X 0,Y 572.938,Z 712,A -85,B 0,C 180,E1 -2250,E2 -2250} C_VEL
LIN {X 0,Y 572.946,Z 711.186,A -85,B 0,C 180,E1 -2251.406,E2 -2251.406} C_VEL
LIN {X 0,Y 572.939,Z 710.2,A -85,B 0,C 180,E1 -2252.109,E2 -2252.109} C_VEL
LIN {X 0,Y 572.959,Z 708.81,A -85,B 0,C 180,E1 -2252.812,E2 -2252.812} C_VEL
LIN {X 0,Y 573.015,Z 705.896,A -85,B 0,C 180,E1 -2253.868,E2 -2253.868} C_VEL
LIN {X 0,Y 572.963,Z 701.949,A -85,B 0,C 180,E1 -2254.926,E2 -2254.926} C_VEL
LIN {X 0,Y 573.064,Z 695.877,A -85,B 0,C 180,E1 -2256.16,E2 -2256.16} C_VEL
LIN {X 0,Y 573.119,Z 689.237,A -85,B 0,C 180,E1 -2257.221,E2 -2257.221} C_VEL
LIN {X 0,Y 573.201,Z 680.99,A -85,B 0,C 180,E1 -2258.283,E2 -2258.283} C_VEL
LIN {X 0,Y 573.287,Z 672.538,A -85,B 0,C 180,E1 -2259.17,E2 -2259.17} C_VEL
LIN {X 0,Y 573.424,Z 662.097,A -85,B 0,C 180,E1 -2260.058,E2 -2260.058} C_VEL
LIN {X 0,Y 573.555,Z 650.401,A -85,B 0,C 180,E1 -2260.855,E2 -2260.855} C_VEL
LIN {X 0,Y 573.653,Z 639.283,A -85,B 0,C 180,E1 -2261.447,E2 -2261.447} C_VEL
LIN {X 0,Y 573.723,Z 626.171,A -85,B 0,C 180,E1 -2261.975,E2 -2261.975} C_VEL
LIN {X 0,Y 573.836,Z 613.517,A -85,B 0,C 180,E1 -2262.331,E2 -2262.331} C_VEL
LIN {X 0,Y 573.896,Z 600.304,A -85,B 0,C 180,E1 -2262.555,E2 -2262.555} C_VEL
LIN {X 0,Y 573.993,Z 502.707,A -85,B 0,C 180,E1 -2263.781,E2 -2263.781} C_VEL
LIN {X 0,Y 573.435,Z 498.452,A -85,B 0,C 180,E1 -2263.872,E2 -2263.872} C_VEL
LIN {X 0,Y 573.687,Z 474.743,A -85,B 0,C 180,E1 -2266.732,E2 -2266.732} C_VEL
LIN {X 0,Y 573.97,Z 450.55,A -85,B 0,C 180,E1 -2269.691,E2 -2269.691} C_VEL
LIN {X 0,Y 574.249,Z 428.078,A -85,B 0,C 180,E1 -2272.486,E2 -2272.486} C_VEL
LIN {X 0,Y 574.46,Z 409.27,A -85,B 0,C 180,E1 -2274.836,E2 -2274.836} C_VEL
LIN {X 0,Y 573.5,Z 403.267,A -85,B 0,C 180,E1 -2275.593,E2 -2275.593} C_VEL
LIN {X 0,Y 573.26,Z 402.082,A -85,B 0,C 180,E1 -2275.751,E2 -2275.751} C_VEL
LIN {X 0,Y 573.207,Z 402.08,A -85,B 0,C 180,E1 -2278.566,E2 -2278.566} C_VEL
LIN {X 0,Y 573.219,Z 402.08,A -85,B 0,C 180,E1 -2280.994,E2 -2280.994} C_VEL
LIN {X 0,Y 573.266,Z 402.081,A -85,B 0,C 180,E1 -2283.524,E2 -2283.524} C_VEL
LIN {X 0,Y 573.191,Z 402.083,A -85,B 0,C 180,E1 -2286.053,E2 -2286.053} C_VEL
LIN {X 0,Y 573.239,Z 402.076,A -85,B 0,C 180,E1 -2288.702,E2 -2288.702} C_VEL
LIN {X 0,Y 573.229,Z 402.082,A -85,B 0,C 180,E1 -2291.593,E2 -2291.593} C_VEL
LIN {X 0,Y 573.228,Z 402.076,A -85,B 0,C 180,E1 -2294.334,E2 -2294.334} C_VEL
LIN {X 0,Y 573.243,Z 402.081,A -85,B 0,C 180,E1 -2297.359,E2 -2297.359} C_VEL
LIN {X 0,Y 573.243,Z 402.075,A -85,B 0,C 180,E1 -2300.392,E2 -2300.392} C_VEL
LIN {X 0,Y 573.255,Z 402.082,A -85,B 0,C 180,E1 -2303.078,E2 -2303.078} C_VEL
LIN {X 0,Y 573.27,Z 402.072,A -85,B 0,C 180,E1 -2305.671,E2 -2305.671} C_VEL
LIN {X 0,Y 573.242,Z 402.075,A -85,B 0,C 180,E1 -2308.185,E2 -2308.185} C_VEL
LIN {X 0,Y 573.263,Z 402.078,A -85,B 0,C 180,E1 -2310.634,E2 -2310.634} C_VEL
LIN {X 0,Y 573.25,Z 402.08,A -85,B 0,C 180,E1 -2313.024,E2 -2313.024} C_VEL
LIN {X 0,Y 573.278,Z 402.072,A -85,B 0,C 180,E1 -2315.366,E2 -2315.366} C_VEL
LIN {X 0,Y 573.231,Z 402.083,A -85,B 0,C 180,E1 -2318.419,E2 -2318.419} C_VEL
LIN {X 0,Y 573.273,Z 402.079,A -85,B 0,C 180,E1 -2320.731,E2 -2320.731} C_VEL
LIN {X 0,Y 573.228,Z 402.078,A -85,B 0,C 180,E1 -2323.621,E2 -2323.621} C_VEL
LIN {X 0,Y 573.198,Z 402.172,A -85,B 0,C 180,E1 -2326.077,E2 -2326.077} C_VEL
LIN {X 0,Y 573.19,Z 402.924,A -85,B 0,C 180,E1 -2326.246,E2 -2326.246} C_VEL
LIN {X 0,Y 574.078,Z 409.093,A -85,B 0,C 180,E1 -2326.347,E2 -2326.347} C_VEL
LIN {X 0,Y 573.866,Z 507.713,A -85,B 0,C 180,E1 -2327.602,E2 -2327.602} C_VEL
LIN {X 0,Y 573.778,Z 520.509,A -85,B 0,C 180,E1 -2327.892,E2 -2327.892} C_VEL
LIN {X 0,Y 573.702,Z 533.342,A -85,B 0,C 180,E1 -2328.339,E2 -2328.339} C_VEL
LIN {X 0,Y 573.584,Z 544.797,A -85,B 0,C 180,E1 -2328.878,E2 -2328.878} C_VEL
LIN {X 0,Y 573.466,Z 555.201,A -85,B 0,C 180,E1 -2329.496,E2 -2329.496} C_VEL
LIN {X 0,Y 573.349,Z 566.016,A -85,B 0,C 180,E1 -2330.297,E2 -2330.297} C_VEL
LIN {X 0,Y 573.241,Z 575.643,A -85,B 0,C 180,E1 -2331.185,E2 -2331.185} C_VEL
LIN {X 0,Y 573.161,Z 583.542,A -85,B 0,C 180,E1 -2332.071,E2 -2332.071} C_VEL
LIN {X 0,Y 573.088,Z 591.572,A -85,B 0,C 180,E1 -2333.169,E2 -2333.169} C_VEL
LIN {X 0,Y 573.07,Z 598.461,A -85,B 0,C 180,E1 -2334.37,E2 -2334.37} C_VEL
LIN {X 0,Y 573.028,Z 603.182,A -85,B 0,C 180,E1 -2335.428,E2 -2335.428} C_VEL
LIN {X 0,Y 573.022,Z 606.803,A -85,B 0,C 180,E1 -2336.484,E2 -2336.484} C_VEL
LIN {X 0,Y 572.959,Z 608.7,A -85,B 0,C 180,E1 -2337.188,E2 -2337.188} C_VEL
LIN {X 0,Y 572.939,Z 610.133,A -85,B 0,C 180,E1 -2337.891,E2 -2337.891} C_VEL
LIN {X 0,Y 572.941,Z 611.758,A -85,B 0,C 180,E1 -2339.297,E2 -2339.297} C_VEL
LIN {X 0,Y 572.939,Z 611.996,A -85,B 0,C 180,E1 -2340,E2 -2340} C_VEL
LIN {X 0,Y 572.947,Z 611.224,A -85,B 0,C 180,E1 -2341.406,E2 -2341.406} C_VEL
LIN {X 0,Y 572.939,Z 610.281,A -85,B 0,C 180,E1 -2342.109,E2 -2342.109} C_VEL
LIN {X 0,Y 572.959,Z 608.885,A -85,B 0,C 180,E1 -2342.812,E2 -2342.812} C_VEL
LIN {X 0,Y 573.015,Z 606.023,A -85,B 0,C 180,E1 -2343.868,E2 -2343.868} C_VEL
LIN {X 0,Y 572.963,Z 602.135,A -85,B 0,C 180,E1 -2344.926,E2 -2344.926} C_VEL
LIN {X 0,Y 573.067,Z 596.108,A -85,B 0,C 180,E1 -2346.16,E2 -2346.16} C_VEL
LIN {X 0,Y 573.114,Z 589.519,A -85,B 0,C 180,E1 -2347.221,E2 -2347.221} C_VEL
LIN {X 0,Y 573.191,Z 581.363,A -85,B 0,C 180,E1 -2348.283,E2 -2348.283} C_VEL
LIN {X 0,Y 573.287,Z 573.008,A -85,B 0,C 180,E1 -2349.17,E2 -2349.17} C_VEL
LIN {X 0,Y 573.423,Z 562.642,A -85,B 0,C 180,E1 -2350.058,E2 -2350.058} C_VEL
LIN {X 0,Y 573.512,Z 552.418,A -85,B 0,C 180,E1 -2350.771,E2 -2350.771} C_VEL
LIN {X 0,Y 573.645,Z 540.333,A -85,B 0,C 180,E1 -2351.443,E2 -2351.443} C_VEL
LIN {X 0,Y 573.727,Z 527.425,A -85,B 0,C 180,E1 -2351.975,E2 -2351.975} C_VEL
LIN {X 0,Y 573.85,Z 515.25,A -85,B 0,C 180,E1 -2352.331,E2 -2352.331} C_VEL
LIN {X 0,Y 573.919,Z 502.083,A -85,B 0,C 180,E1 -2352.577,E2 -2352.577} C_VEL
LIN {X 0,Y 574.066,Z 428.061,A -85,B 0,C 180,E1 -2353.504,E2 -2353.504} C_VEL
LIN {X 0,Y 573.469,Z 424.199,A -85,B 0,C 180,E1 -2353.567,E2 -2353.567} C_VEL
LIN {X 0,Y 570.912,Z 418.185,A -85,B 0,C 180,E1 -2353.705,E2 -2353.705} C_VEL
LIN {X 0,Y 567.658,Z 410.959,A -85,B 0,C 180,E1 -2353.877,E2 -2353.877} C_VEL
LIN {X 0,Y 567.077,Z 408.38,A -85,B 0,C 180,E1 -2353.925,E2 -2353.925} C_VEL
LIN {X 0,Y 566.14,Z 402.965,A -85,B 0,C 180,E1 -2354.032,E2 -2354.032} C_VEL
LIN {X 0,Y 566.168,Z 402.957,A -85,B 0,C 180,E1 -2356.589,E2 -2356.589} C_VEL
LIN {X 0,Y 566.204,Z 402.961,A -85,B 0,C 180,E1 -2359.581,E2 -2359.581} C_VEL
LIN {X 0,Y 566.191,Z 402.956,A -85,B 0,C 180,E1 -2361.863,E2 -2361.863} C_VEL
LIN {X 0,Y 566.185,Z 402.957,A -85,B 0,C 180,E1 -2365.022,E2 -2365.022} C_VEL
LIN {X 0,Y 566.193,Z 402.96,A -85,B 0,C 180,E1 -2367.34,E2 -2367.34} C_VEL
LIN {X 0,Y 566.203,Z 402.953,A -85,B 0,C 180,E1 -2369.769,E2 -2369.769} C_VEL
LIN {X 0,Y 566.205,Z 402.95,A -85,B 0,C 180,E1 -2372.43,E2 -2372.43} C_VEL
LIN {X 0,Y 566.183,Z 402.959,A -85,B 0,C 180,E1 -2374.989,E2 -2374.989} C_VEL
LIN {X 0,Y 566.2,Z 402.955,A -85,B 0,C 180,E1 -2377.461,E2 -2377.461} C_VEL
LIN {X 0,Y 566.211,Z 402.949,A -85,B 0,C 180,E1 -2380.199,E2 -2380.199} C_VEL
LIN {X 0,Y 566.204,Z 402.958,A -85,B 0,C 180,E1 -2383.054,E2 -2383.054} C_VEL
LIN {X 0,Y 566.202,Z 402.95,A -85,B 0,C 180,E1 -2386.049,E2 -2386.049} C_VEL
LIN {X 0,Y 566.207,Z 402.952,A -85,B 0,C 180,E1 -2389.215,E2 -2389.215} C_VEL
LIN {X 0,Y 566.184,Z 402.954,A -85,B 0,C 180,E1 -2391.636,E2 -2391.636} C_VEL
LIN {X 0,Y 566.152,Z 402.963,A -85,B 0,C 180,E1 -2394.307,E2 -2394.307} C_VEL
LIN {X 0,Y 566.222,Z 402.953,A -85,B 0,C 180,E1 -2396.898,E2 -2396.898} C_VEL
LIN {X 0,Y 566.172,Z 402.956,A -85,B 0,C 180,E1 -2399.407,E2 -2399.407} C_VEL
LIN {X 0,Y 566.173,Z 402.959,A -85,B 0,C 180,E1 -2401.855,E2 -2401.855} C_VEL
LIN {X 0,Y 566.189,Z 402.963,A -85,B 0,C 180,E1 -2404.25,E2 -2404.25} C_VEL
LIN {X 0,Y 566.198,Z 403.043,A -85,B 0,C 180,E1 -2406.403,E2 -2406.403} C_VEL
LIN {X 0,Y 567.109,Z 408.439,A -85,B 0,C 180,E1 -2407.215,E2 -2407.215} C_VEL
LIN {X 0,Y 566.885,Z 428.045,A -85,B 0,C 180,E1 -2410.067,E2 -2410.067} C_VEL
LIN {X 0,Y 566.612,Z 447.631,A -85,B 0,C 180,E1 -2412.893,E2 -2412.893} C_VEL
LIN {X 0,Y 566.39,Z 469.618,A -85,B 0,C 180,E1 -2416.02,E2 -2416.02} C_VEL
LIN {X 0,Y 567.144,Z 475.558,A -85,B 0,C 180,E1 -2416.131,E2 -2416.131} C_VEL
LIN {X 0,Y 566.939,Z 577.66,A -85,B 0,C 180,E1 -2417.448,E2 -2417.448} C_VEL
LIN {X 0,Y 566.85,Z 588.752,A -85,B 0,C 180,E1 -2417.696,E2 -2417.696} C_VEL
LIN {X 0,Y 566.751,Z 601.152,A -85,B 0,C 180,E1 -2418.103,E2 -2418.103} C_VEL
LIN {X 0,Y 566.627,Z 614.389,A -85,B 0,C 180,E1 -2418.714,E2 -2418.714} C_VEL
LIN {X 0,Y 566.495,Z 625.181,A -85,B 0,C 180,E1 -2419.366,E2 -2419.366} C_VEL
LIN {X 0,Y 566.317,Z 634.868,A -85,B 0,C 180,E1 -2420.085,E2 -2420.085} C_VEL
LIN {X 0,Y 566.237,Z 643.847,A -85,B 0,C 180,E1 -2420.895,E2 -2420.895} C_VEL
LIN {X 0,Y 566.127,Z 652.1,A -85,B 0,C 180,E1 -2421.792,E2 -2421.792} C_VEL
LIN {X 0,Y 566.041,Z 660.169,A -85,B 0,C 180,E1 -2422.868,E2 -2422.868} C_VEL
LIN {X 0,Y 566.003,Z 666.617,A -85,B 0,C 180,E1 -2423.941,E2 -2423.941} C_VEL
LIN {X 0,Y 565.877,Z 671.735,A -85,B 0,C 180,E1 -2425.013,E2 -2425.013} C_VEL
LIN {X 0,Y 565.926,Z 675.718,A -85,B 0,C 180,E1 -2426.084,E2 -2426.084} C_VEL
LIN {X 0,Y 565.877,Z 678.673,A -85,B 0,C 180,E1 -2427.152,E2 -2427.152} C_VEL
LIN {X 0,Y 565.84,Z 680.138,A -85,B 0,C 180,E1 -2427.865,E2 -2427.865} C_VEL
LIN {X 0,Y 565.841,Z 681.747,A -85,B 0,C 180,E1 -2429.288,E2 -2429.288} C_VEL
LIN {X 0,Y 565.839,Z 681.996,A -85,B 0,C 180,E1 -2430,E2 -2430} C_VEL
LIN {X 0,Y 565.846,Z 681.23,A -85,B 0,C 180,E1 -2431.423,E2 -2431.423} C_VEL
LIN {X 0,Y 565.84,Z 680.279,A -85,B 0,C 180,E1 -2432.135,E2 -2432.135} C_VEL
LIN {X 0,Y 565.927,Z 677.067,A -85,B 0,C 180,E1 -2433.56,E2 -2433.56} C_VEL
LIN {X 0,Y 565.933,Z 673.511,A -85,B 0,C 180,E1 -2434.63,E2 -2434.63} C_VEL
LIN {X 0,Y 565.998,Z 668.863,A -85,B 0,C 180,E1 -2435.701,E2 -2435.701} C_VEL
LIN {X 0,Y 565.999,Z 663.197,A -85,B 0,C 180,E1 -2436.739,E2 -2436.739} C_VEL
LIN {X 0,Y 566.095,Z 655.669,A -85,B 0,C 180,E1 -2437.849,E2 -2437.849} C_VEL
LIN {X 0,Y 566.202,Z 646.55,A -85,B 0,C 180,E1 -2438.926,E2 -2438.926} C_VEL
LIN {X 0,Y 566.324,Z 637.053,A -85,B 0,C 180,E1 -2439.825,E2 -2439.825} C_VEL
LIN {X 0,Y 566.445,Z 627.795,A -85,B 0,C 180,E1 -2440.545,E2 -2440.545} C_VEL
LIN {X 0,Y 566.579,Z 618.435,A -85,B 0,C 180,E1 -2441.146,E2 -2441.146} C_VEL
LIN {X 0,Y 566.678,Z 609.36,A -85,B 0,C 180,E1 -2441.626,E2 -2441.626} C_VEL
LIN {X 0,Y 566.723,Z 598.609,A -85,B 0,C 180,E1 -2442.079,E2 -2442.079} C_VEL
LIN {X 0,Y 566.887,Z 587.857,A -85,B 0,C 180,E1 -2442.417,E2 -2442.417} C_VEL
LIN {X 0,Y 566.949,Z 577.604,A -85,B 0,C 180,E1 -2442.643,E2 -2442.643} C_VEL
LIN {X 0,Y 567.054,Z 474.327,A -85,B 0,C 180,E1 -2443.977,E2 -2443.977} C_VEL
LIN {X 0,Y 566.412,Z 469.607,A -85,B 0,C 180,E1 -2444.071,E2 -2444.071} C_VEL
LIN {X 0,Y 566.612,Z 448.257,A -85,B 0,C 180,E1 -2447.107,E2 -2447.107} C_VEL
LIN {X 0,Y 566.911,Z 427.364,A -85,B 0,C 180,E1 -2450.122,E2 -2450.122} C_VEL
LIN {X 0,Y 567.099,Z 409.087,A -85,B 0,C 180,E1 -2452.785,E2 -2452.785} C_VEL
LIN {X 0,Y 566.171,Z 402.965,A -85,B 0,C 180,E1 -2453.72,E2 -2453.72} C_VEL
LIN {X 0,Y 566.171,Z 402.957,A -85,B 0,C 180,E1 -2456.651,E2 -2456.651} C_VEL
LIN {X 0,Y 566.175,Z 402.964,A -85,B 0,C 180,E1 -2459.666,E2 -2459.666} C_VEL
LIN {X 0,Y 566.203,Z 402.952,A -85,B 0,C 180,E1 -2462.429,E2 -2462.429} C_VEL
LIN {X 0,Y 566.18,Z 402.958,A -85,B 0,C 180,E1 -2464.989,E2 -2464.989} C_VEL
LIN {X 0,Y 566.195,Z 402.96,A -85,B 0,C 180,E1 -2467.461,E2 -2467.461} C_VEL
LIN {X 0,Y 566.21,Z 402.949,A -85,B 0,C 180,E1 -2470.199,E2 -2470.199} C_VEL
LIN {X 0,Y 566.205,Z 402.96,A -85,B 0,C 180,E1 -2473.054,E2 -2473.054} C_VEL
LIN {X 0,Y 566.202,Z 402.952,A -85,B 0,C 180,E1 -2476.049,E2 -2476.049} C_VEL
LIN {X 0,Y 566.207,Z 402.955,A -85,B 0,C 180,E1 -2479.215,E2 -2479.215} C_VEL
LIN {X 0,Y 566.189,Z 402.953,A -85,B 0,C 180,E1 -2481.637,E2 -2481.637} C_VEL
LIN {X 0,Y 566.153,Z 402.958,A -85,B 0,C 180,E1 -2484.307,E2 -2484.307} C_VEL
LIN {X 0,Y 566.222,Z 402.954,A -85,B 0,C 180,E1 -2486.898,E2 -2486.898} C_VEL
LIN {X 0,Y 566.173,Z 402.955,A -85,B 0,C 180,E1 -2489.407,E2 -2489.407} C_VEL
LIN {X 0,Y 566.173,Z 402.958,A -85,B 0,C 180,E1 -2491.855,E2 -2491.855} C_VEL
LIN {X 0,Y 566.194,Z 402.961,A -85,B 0,C 180,E1 -2494.25,E2 -2494.25} C_VEL
LIN {X 0,Y 566.195,Z 403.066,A -85,B 0,C 180,E1 -2496.378,E2 -2496.378} C_VEL
LIN {X 0,Y 567.105,Z 408.523,A -85,B 0,C 180,E1 -2497.215,E2 -2497.215} C_VEL
LIN {X 0,Y 566.891,Z 428.042,A -85,B 0,C 180,E1 -2500.066,E2 -2500.066} C_VEL
LIN {X 0,Y 566.612,Z 447.63,A -85,B 0,C 180,E1 -2502.893,E2 -2502.893} C_VEL
LIN {X 0,Y 566.394,Z 469.618,A -85,B 0,C 180,E1 -2506.02,E2 -2506.02} C_VEL
LIN {X 0,Y 567.146,Z 475.556,A -85,B 0,C 180,E1 -2506.131,E2 -2506.131} C_VEL
LIN {X 0,Y 566.939,Z 577.697,A -85,B 0,C 180,E1 -2507.448,E2 -2507.448} C_VEL
LIN {X 0,Y 566.837,Z 589.682,A -85,B 0,C 180,E1 -2507.718,E2 -2507.718} C_VEL
LIN {X 0,Y 566.697,Z 603.381,A -85,B 0,C 180,E1 -2508.193,E2 -2508.193} C_VEL
LIN {X 0,Y 566.637,Z 614.474,A -85,B 0,C 180,E1 -2508.722,E2 -2508.722} C_VEL
LIN {X 0,Y 566.502,Z 623.814,A -85,B 0,C 180,E1 -2509.275,E2 -2509.275} C_VEL
LIN {X 0,Y 566.35,Z 633.77,A -85,B 0,C 180,E1 -2509.995,E2 -2509.995} C_VEL
LIN {X 0,Y 566.238,Z 643.91,A -85,B 0,C 180,E1 -2510.895,E2 -2510.895} C_VEL
LIN {X 0,Y 566.113,Z 653.551,A -85,B 0,C 180,E1 -2511.972,E2 -2511.972} C_VEL
LIN {X 0,Y 566.05,Z 660.124,A -85,B 0,C 180,E1 -2512.868,E2 -2512.868} C_VEL
LIN {X 0,Y 565.992,Z 666.573,A -85,B 0,C 180,E1 -2513.941,E2 -2513.941} C_VEL
LIN {X 0,Y 565.877,Z 671.721,A -85,B 0,C 180,E1 -2515.012,E2 -2515.012} C_VEL
LIN {X 0,Y 565.926,Z 675.717,A -85,B 0,C 180,E1 -2516.083,E2 -2516.083} C_VEL
LIN {X 0,Y 565.877,Z 678.677,A -85,B 0,C 180,E1 -2517.152,E2 -2517.152} C_VEL
LIN {X 0,Y 565.845,Z 681.142,A -85,B 0,C 180,E1 -2518.577,E2 -2518.577} C_VEL
LIN {X 0,Y 565.841,Z 681.753,A -85,B 0,C 180,E1 -2519.288,E2 -2519.288} C_VEL
LIN {X 0,Y 565.841,Z 681.81,A -85,B 0,C 180,E1 -2520.712,E2 -2520.712} C_VEL
LIN {X 0,Y 565.846,Z 681.241,A -85,B 0,C 180,E1 -2521.423,E2 -2521.423} C_VEL
LIN {X 0,Y 565.878,Z 678.898,A -85,B 0,C 180,E1 -2522.848,E2 -2522.848} C_VEL
LIN {X 0,Y 565.927,Z 676.024,A -85,B 0,C 180,E1 -2523.916,E2 -2523.916} C_VEL
LIN {X 0,Y 565.878,Z 672.114,A -85,B 0,C 180,E1 -2524.987,E2 -2524.987} C_VEL
LIN {X 0,Y 565.994,Z 667.06,A -85,B 0,C 180,E1 -2526.059,E2 -2526.059} C_VEL
LIN {X 0,Y 566.032,Z 660.713,A -85,B 0,C 180,E1 -2527.132,E2 -2527.132} C_VEL
LIN {X 0,Y 566.128,Z 652.857,A -85,B 0,C 180,E1 -2528.208,E2 -2528.208} C_VEL
LIN {X 0,Y 566.249,Z 642.979,A -85,B 0,C 180,E1 -2529.285,E2 -2529.285} C_VEL
LIN {X 0,Y 566.405,Z 633.766,A -85,B 0,C 180,E1 -2530.094,E2 -2530.094} C_VEL
LIN {X 0,Y 566.506,Z 623.918,A -85,B 0,C 180,E1 -2530.808,E2 -2530.808} C_VEL
LIN {X 0,Y 566.661,Z 613.047,A -85,B 0,C 180,E1 -2531.446,E2 -2531.446} C_VEL
LIN {X 0,Y 566.72,Z 599.948,A -85,B 0,C 180,E1 -2532.034,E2 -2532.034} C_VEL
LIN {X 0,Y 566.887,Z 587.886,A -85,B 0,C 180,E1 -2532.417,E2 -2532.417} C_VEL
LIN {X 0,Y 566.949,Z 577.643,A -85,B 0,C 180,E1 -2532.643,E2 -2532.643} C_VEL
LIN {X 0,Y 567.052,Z 474.33,A -85,B 0,C 180,E1 -2533.977,E2 -2533.977} C_VEL
LIN {X 0,Y 566.406,Z 469.607,A -85,B 0,C 180,E1 -2534.071,E2 -2534.071} C_VEL
LIN {X 0,Y 566.611,Z 448.258,A -85,B 0,C 180,E1 -2537.107,E2 -2537.107} C_VEL
LIN {X 0,Y 566.911,Z 427.366,A -85,B 0,C 180,E1 -2540.122,E2 -2540.122} C_VEL
LIN {X 0,Y 567.121,Z 410.341,A -85,B 0,C 180,E1 -2542.592,E2 -2542.592} C_VEL
LIN {X 0,Y 566.538,Z 404.812,A -85,B 0,C 180,E1 -2543.389,E2 -2543.389} C_VEL
LIN {X 0,Y 566.181,Z 402.963,A -85,B 0,C 180,E1 -2543.695,E2 -2543.695} C_VEL
LIN {X 0,Y 566.171,Z 402.957,A -85,B 0,C 180,E1 -2546.651,E2 -2546.651} C_VEL
LIN {X 0,Y 566.175,Z 402.965,A -85,B 0,C 180,E1 -2549.666,E2 -2549.666} C_VEL
LIN {X 0,Y 566.203,Z 402.952,A -85,B 0,C 180,E1 -2552.429,E2 -2552.429} C_VEL
LIN {X 0,Y 566.18,Z 402.958,A -85,B 0,C 180,E1 -2554.989,E2 -2554.989} C_VEL
LIN {X 0,Y 566.195,Z 402.96,A -85,B 0,C 180,E1 -2557.461,E2 -2557.461} C_VEL
LIN {X 0,Y 566.21,Z 402.951,A -85,B 0,C 180,E1 -2560.199,E2 -2560.199} C_VEL
LIN {X 0,Y 566.204,Z 402.96,A -85,B 0,C 180,E1 -2563.054,E2 -2563.054} C_VEL
LIN {X 0,Y 566.202,Z 402.952,A -85,B 0,C 180,E1 -2566.049,E2 -2566.049} C_VEL
LIN {X 0,Y 566.207,Z 402.955,A -85,B 0,C 180,E1 -2569.215,E2 -2569.215} C_VEL
LIN {X 0,Y 566.186,Z 402.954,A -85,B 0,C 180,E1 -2571.637,E2 -2571.637} C_VEL
LIN {X 0,Y 566.152,Z 402.962,A -85,B 0,C 180,E1 -2574.307,E2 -2574.307} C_VEL
LIN {X 0,Y 566.222,Z 402.954,A -85,B 0,C 180,E1 -2576.898,E2 -2576.898} C_VEL
LIN {X 0,Y 566.172,Z 402.956,A -85,B 0,C 180,E1 -2579.407,E2 -2579.407} C_VEL
LIN {X 0,Y 566.172,Z 402.959,A -85,B 0,C 180,E1 -2581.855,E2 -2581.855} C_VEL
LIN {X 0,Y 566.206,Z 403.021,A -85,B 0,C 180,E1 -2584.053,E2 -2584.053} C_VEL
LIN {X 0,Y 567.478,Z 409.078,A -85,B 0,C 180,E1 -2584.871,E2 -2584.871} C_VEL
LIN {X 0,Y 567.435,Z 428.029,A -85,B 0,C 180,E1 -2587.229,E2 -2587.229} C_VEL
LIN {X 0,Y 567.076,Z 449.303,A -85,B 0,C 180,E1 -2589.903,E2 -2589.903} C_VEL
LIN {X 0,Y 566.744,Z 473.06,A -85,B 0,C 180,E1 -2592.849,E2 -2592.849} C_VEL
LIN {X 0,Y 566.471,Z 498.075,A -85,B 0,C 180,E1 -2595.908,E2 -2595.908} C_VEL
LIN {X 0,Y 566.458,Z 498.64,A -85,B 0,C 180,E1 -2595.976,E2 -2595.976} C_VEL
LIN {X 0,Y 567.162,Z 505.502,A -85,B 0,C 180,E1 -2596.085,E2 -2596.085} C_VEL
LIN {X 0,Y 566.972,Z 607.943,A -85,B 0,C 180,E1 -2597.403,E2 -2597.403} C_VEL
LIN {X 0,Y 566.847,Z 621.216,A -85,B 0,C 180,E1 -2597.719,E2 -2597.719} C_VEL
LIN {X 0,Y 566.736,Z 632.917,A -85,B 0,C 180,E1 -2598.13,E2 -2598.13} C_VEL
LIN {X 0,Y 566.63,Z 645.063,A -85,B 0,C 180,E1 -2598.703,E2 -2598.703} C_VEL
LIN {X 0,Y 566.5,Z 655.908,A -85,B 0,C 180,E1 -2599.366,E2 -2599.366} C_VEL
LIN {X 0,Y 566.336,Z 666.54,A -85,B 0,C 180,E1 -2600.175,E2 -2600.175} C_VEL
LIN {X 0,Y 566.207,Z 676.112,A -85,B 0,C 180,E1 -2601.074,E2 -2601.074} C_VEL
LIN {X 0,Y 566.112,Z 683.96,A -85,B 0,C 180,E1 -2601.972,E2 -2601.972} C_VEL
LIN {X 0,Y 566.003,Z 691.621,A -85,B 0,C 180,E1 -2603.047,E2 -2603.047} C_VEL
LIN {X 0,Y 566.004,Z 698.68,A -85,B 0,C 180,E1 -2604.299,E2 -2604.299} C_VEL
LIN {X 0,Y 565.933,Z 703.372,A -85,B 0,C 180,E1 -2605.37,E2 -2605.37} C_VEL
LIN {X 0,Y 565.927,Z 706.957,A -85,B 0,C 180,E1 -2606.44,E2 -2606.44} C_VEL
LIN {X 0,Y 565.878,Z 708.808,A -85,B 0,C 180,E1 -2607.152,E2 -2607.152} C_VEL
LIN {X 0,Y 565.846,Z 711.185,A -85,B 0,C 180,E1 -2608.577,E2 -2608.577} C_VEL
LIN {X 0,Y 565.839,Z 712,A -85,B 0,C 180,E1 -2610,E2 -2610} C_VEL
LIN {X 0,Y 565.846,Z 711.186,A -85,B 0,C 180,E1 -2611.423,E2 -2611.423} C_VEL
LIN {X 0,Y 565.878,Z 708.81,A -85,B 0,C 180,E1 -2612.848,E2 -2612.848} C_VEL
LIN {X 0,Y 565.926,Z 705.896,A -85,B 0,C 180,E1 -2613.916,E2 -2613.916} C_VEL
LIN {X 0,Y 565.878,Z 701.949,A -85,B 0,C 180,E1 -2614.987,E2 -2614.987} C_VEL
LIN {X 0,Y 566.002,Z 696.867,A -85,B 0,C 180,E1 -2616.059,E2 -2616.059} C_VEL
LIN {X 0,Y 566.04,Z 690.468,A -85,B 0,C 180,E1 -2617.132,E2 -2617.132} C_VEL
LIN {X 0,Y 566.134,Z 682.478,A -85,B 0,C 180,E1 -2618.208,E2 -2618.208} C_VEL
LIN {X 0,Y 566.229,Z 674.335,A -85,B 0,C 180,E1 -2619.106,E2 -2619.106} C_VEL
LIN {X 0,Y 566.345,Z 664.4,A -85,B 0,C 180,E1 -2620.005,E2 -2620.005} C_VEL
LIN {X 0,Y 566.529,Z 653.301,A -85,B 0,C 180,E1 -2620.807,E2 -2620.807} C_VEL
LIN {X 0,Y 566.613,Z 642.175,A -85,B 0,C 180,E1 -2621.447,E2 -2621.447} C_VEL
LIN {X 0,Y 566.721,Z 629.982,A -85,B 0,C 180,E1 -2621.989,E2 -2621.989} C_VEL
LIN {X 0,Y 566.881,Z 617.173,A -85,B 0,C 180,E1 -2622.394,E2 -2622.394} C_VEL
LIN {X 0,Y 566.938,Z 605.101,A -85,B 0,C 180,E1 -2622.643,E2 -2622.643} C_VEL
LIN {X 0,Y 567.047,Z 502.944,A -85,B 0,C 180,E1 -2623.95,E2 -2623.95} C_VEL
LIN {X 0,Y 566.458,Z 498.452,A -85,B 0,C 180,E1 -2624.047,E2 -2624.047} C_VEL
LIN {X 0,Y 566.724,Z 475.049,A -85,B 0,C 180,E1 -2626.906,E2 -2626.906} C_VEL
LIN {X 0,Y 567.049,Z 452.315,A -85,B 0,C 180,E1 -2629.72,E2 -2629.72} C_VEL
LIN {X 0,Y 567.335,Z 432.594,A -85,B 0,C 180,E1 -2632.199,E2 -2632.199} C_VEL
LIN {X 0,Y 567.5,Z 410.504,A -85,B 0,C 180,E1 -2634.902,E2 -2634.902} C_VEL
LIN {X 0,Y 566.391,Z 403.954,A -85,B 0,C 180,E1 -2635.74,E2 -2635.74} C_VEL
LIN {X 0,Y 566.213,Z 402.959,A -85,B 0,C 180,E1 -2635.897,E2 -2635.897} C_VEL
LIN {X 0,Y 566.165,Z 402.959,A -85,B 0,C 180,E1 -2638.955,E2 -2638.955} C_VEL
LIN {X 0,Y 566.19,Z 402.961,A -85,B 0,C 180,E1 -2641.422,E2 -2641.422} C_VEL
LIN {X 0,Y 566.21,Z 402.955,A -85,B 0,C 180,E1 -2643.956,E2 -2643.956} C_VEL
LIN {X 0,Y 566.195,Z 402.961,A -85,B 0,C 180,E1 -2647.4,E2 -2647.4} C_VEL
LIN {X 0,Y 566.209,Z 402.951,A -85,B 0,C 180,E1 -2650.199,E2 -2650.199} C_VEL
LIN {X 0,Y 566.199,Z 402.957,A -85,B 0,C 180,E1 -2653.055,E2 -2653.055} C_VEL
LIN {X 0,Y 566.201,Z 402.952,A -85,B 0,C 180,E1 -2656.049,E2 -2656.049} C_VEL
LIN {X 0,Y 566.207,Z 402.959,A -85,B 0,C 180,E1 -2659.215,E2 -2659.215} C_VEL
LIN {X 0,Y 566.189,Z 402.955,A -85,B 0,C 180,E1 -2661.637,E2 -2661.637} C_VEL
LIN {X 0,Y 566.166,Z 402.957,A -85,B 0,C 180,E1 -2664.308,E2 -2664.308} C_VEL
LIN {X 0,Y 566.223,Z 402.958,A -85,B 0,C 180,E1 -2666.898,E2 -2666.898} C_VEL
LIN {X 0,Y 566.183,Z 402.956,A -85,B 0,C 180,E1 -2669.407,E2 -2669.407} C_VEL
LIN {X 0,Y 566.215,Z 402.95,A -85,B 0,C 180,E1 -2671.857,E2 -2671.857} C_VEL
LIN {X 0,Y 566.209,Z 402.954,A -85,B 0,C 180,E1 -2674.251,E2 -2674.251} C_VEL
LIN {X 0,Y 566.176,Z 402.965,A -85,B 0,C 180,E1 -2676.718,E2 -2676.718} C_VEL
LIN {X 0,Y 566.207,Z 402.952,A -85,B 0,C 180,E1 -2679.663,E2 -2679.663} C_VEL
LIN {X 0,Y 566.194,Z 402.961,A -85,B 0,C 180,E1 -2682.668,E2 -2682.668} C_VEL
LIN {X 0,Y 566.213,Z 402.953,A -85,B 0,C 180,E1 -2685.626,E2 -2685.626} C_VEL
LIN {X 0,Y 566.16,Z 402.964,A -85,B 0,C 180,E1 -2686.072,E2 -2686.072} C_VEL
LIN {X 0,Y 567.198,Z 409.138,A -85,B 0,C 180,E1 -2686.178,E2 -2686.178} C_VEL
LIN {X 0,Y 566.951,Z 507.698,A -85,B 0,C 180,E1 -2687.448,E2 -2687.448} C_VEL
LIN {X 0,Y 566.856,Z 520.538,A -85,B 0,C 180,E1 -2687.742,E2 -2687.742} C_VEL
LIN {X 0,Y 566.732,Z 533.334,A -85,B 0,C 180,E1 -2688.193,E2 -2688.193} C_VEL
LIN {X 0,Y 566.629,Z 544.296,A -85,B 0,C 180,E1 -2688.713,E2 -2688.713} C_VEL
LIN {X 0,Y 566.508,Z 553.804,A -85,B 0,C 180,E1 -2689.275,E2 -2689.275} C_VEL
LIN {X 0,Y 566.35,Z 563.791,A -85,B 0,C 180,E1 -2689.995,E2 -2689.995} C_VEL
LIN {X 0,Y 566.238,Z 573.902,A -85,B 0,C 180,E1 -2690.895,E2 -2690.895} C_VEL
LIN {X 0,Y 566.134,Z 582.1,A -85,B 0,C 180,E1 -2691.792,E2 -2691.792} C_VEL
LIN {X 0,Y 566.053,Z 588.899,A -85,B 0,C 180,E1 -2692.689,E2 -2692.689} C_VEL
LIN {X 0,Y 565.989,Z 595.589,A -85,B 0,C 180,E1 -2693.762,E2 -2693.762} C_VEL
LIN {X 0,Y 565.937,Z 600.134,A -85,B 0,C 180,E1 -2694.656,E2 -2694.656} C_VEL
LIN {X 0,Y 565.959,Z 604.512,A -85,B 0,C 180,E1 -2695.727,E2 -2695.727} C_VEL
LIN {X 0,Y 565.877,Z 608.698,A -85,B 0,C 180,E1 -2697.152,E2 -2697.152} C_VEL
LIN {X 0,Y 565.84,Z 610.131,A -85,B 0,C 180,E1 -2697.865,E2 -2697.865} C_VEL
LIN {X 0,Y 565.841,Z 611.753,A -85,B 0,C 180,E1 -2699.288,E2 -2699.288} C_VEL
LIN {X 0,Y 565.839,Z 611.996,A -85,B 0,C 180,E1 -2700,E2 -2700} C_VEL
LIN {X 0,Y 565.846,Z 611.218,A -85,B 0,C 180,E1 -2701.423,E2 -2701.423} C_VEL
LIN {X 0,Y 565.84,Z 610.282,A -85,B 0,C 180,E1 -2702.135,E2 -2702.135} C_VEL
LIN {X 0,Y 565.878,Z 608.878,A -85,B 0,C 180,E1 -2702.848,E2 -2702.848} C_VEL
LIN {X 0,Y 565.959,Z 604.841,A -85,B 0,C 180,E1 -2704.273,E2 -2704.273} C_VEL
LIN {X 0,Y 565.936,Z 600.557,A -85,B 0,C 180,E1 -2705.344,E2 -2705.344} C_VEL
LIN {X 0,Y 565.966,Z 595.084,A -85,B 0,C 180,E1 -2706.417,E2 -2706.417} C_VEL
LIN {X 0,Y 566.054,Z 588.287,A -85,B 0,C 180,E1 -2707.491,E2 -2707.491} C_VEL
LIN {X 0,Y 566.165,Z 579.824,A -85,B 0,C 180,E1 -2708.567,E2 -2708.567} C_VEL
LIN {X 0,Y 566.281,Z 571.065,A -85,B 0,C 180,E1 -2709.465,E2 -2709.465} C_VEL
LIN {X 0,Y 566.426,Z 561.447,A -85,B 0,C 180,E1 -2710.274,E2 -2710.274} C_VEL
LIN {X 0,Y 566.559,Z 551.27,A -85,B 0,C 180,E1 -2710.977,E2 -2710.977} C_VEL
LIN {X 0,Y 566.69,Z 538.778,A -85,B 0,C 180,E1 -2711.658,E2 -2711.658} C_VEL
LIN {X 0,Y 566.782,Z 527.385,A -85,B 0,C 180,E1 -2712.124,E2 -2712.124} C_VEL
LIN {X 0,Y 566.898,Z 516.105,A -85,B 0,C 180,E1 -2712.462,E2 -2712.462} C_VEL
LIN {X 0,Y 566.987,Z 503.562,A -85,B 0,C 180,E1 -2712.71,E2 -2712.71} C_VEL
LIN {X 0,Y 567.077,Z 408.38,A -85,B 0,C 180,E1 -2713.925,E2 -2713.925} C_VEL
LIN {X 0,Y 566.501,Z 406.283,A -85,B 0,C 180,E1 -2714.033,E2 -2714.033} C_VEL
LIN {X 0,Y 565.356,Z 404.493,A -85,B 0,C 180,E1 -2714.299,E2 -2714.299} C_VEL
LIN {X 0,Y 563.723,Z 403.533,A -85,B 0,C 180,E1 -2714.732,E2 -2714.732} C_VEL
LIN {X 0,Y 561.224,Z 403.581,A -85,B 0,C 180,E1 -2715.559,E2 -2715.559} C_VEL
LIN {X 0,Y 559.416,Z 403.803,A -85,B 0,C 180,E1 -2716.493,E2 -2716.493} C_VEL
LIN {X 0,Y 559.146,Z 403.833,A -85,B 0,C 180,E1 -2716.968,E2 -2716.968} C_VEL
LIN {X 0,Y 559.167,Z 403.833,A -85,B 0,C 180,E1 -2719.838,E2 -2719.838} C_VEL
LIN {X 0,Y 559.139,Z 403.831,A -85,B 0,C 180,E1 -2722.153,E2 -2722.153} C_VEL
LIN {X 0,Y 559.144,Z 403.837,A -85,B 0,C 180,E1 -2725.178,E2 -2725.178} C_VEL
LIN {X 0,Y 559.141,Z 403.833,A -85,B 0,C 180,E1 -2727.714,E2 -2727.714} C_VEL
LIN {X 0,Y 559.156,Z 403.829,A -85,B 0,C 180,E1 -2730.183,E2 -2730.183} C_VEL
LIN {X 0,Y 559.159,Z 403.83,A -85,B 0,C 180,E1 -2732.715,E2 -2732.715} C_VEL
LIN {X 0,Y 559.131,Z 403.838,A -85,B 0,C 180,E1 -2735.324,E2 -2735.324} C_VEL
LIN {X 0,Y 559.137,Z 403.832,A -85,B 0,C 180,E1 -2738.018,E2 -2738.018} C_VEL
LIN {X 0,Y 559.159,Z 403.834,A -85,B 0,C 180,E1 -2740.812,E2 -2740.812} C_VEL
LIN {X 0,Y 559.144,Z 403.831,A -85,B 0,C 180,E1 -2743.734,E2 -2743.734} C_VEL
LIN {X 0,Y 559.17,Z 403.835,A -85,B 0,C 180,E1 -2746.801,E2 -2746.801} C_VEL
LIN {X 0,Y 559.159,Z 403.83,A -85,B 0,C 180,E1 -2749.188,E2 -2749.188} C_VEL
LIN {X 0,Y 559.132,Z 403.834,A -85,B 0,C 180,E1 -2751.982,E2 -2751.982} C_VEL
LIN {X 0,Y 559.131,Z 403.838,A -85,B 0,C 180,E1 -2754.788,E2 -2754.788} C_VEL
LIN {X 0,Y 559.158,Z 403.829,A -85,B 0,C 180,E1 -2757.365,E2 -2757.365} C_VEL
LIN {X 0,Y 559.124,Z 403.84,A -85,B 0,C 180,E1 -2760.148,E2 -2760.148} C_VEL
LIN {X 0,Y 559.119,Z 403.836,A -85,B 0,C 180,E1 -2763.184,E2 -2763.184} C_VEL
LIN {X 0,Y 559.141,Z 403.841,A -85,B 0,C 180,E1 -2766.185,E2 -2766.185} C_VEL
LIN {X 0,Y 559.156,Z 403.984,A -85,B 0,C 180,E1 -2766.284,E2 -2766.284} C_VEL
LIN {X 0,Y 560.129,Z 409.419,A -85,B 0,C 180,E1 -2767.11,E2 -2767.11} C_VEL
LIN {X 0,Y 559.943,Z 429.331,A -85,B 0,C 180,E1 -2770,E2 -2770} C_VEL
LIN {X 0,Y 559.626,Z 449.362,A -85,B 0,C 180,E1 -2772.924,E2 -2772.924} C_VEL
LIN {X 0,Y 559.389,Z 469.622,A -85,B 0,C 180,E1 -2775.842,E2 -2775.842} C_VEL
LIN {X 0,Y 560.245,Z 475.604,A -85,B 0,C 180,E1 -2775.956,E2 -2775.956} C_VEL
LIN {X 0,Y 560.009,Z 577.641,A -85,B 0,C 180,E1 -2777.29,E2 -2777.29} C_VEL
LIN {X 0,Y 559.917,Z 588.741,A -85,B 0,C 180,E1 -2777.541,E2 -2777.541} C_VEL
LIN {X 0,Y 559.791,Z 601.152,A -85,B 0,C 180,E1 -2777.953,E2 -2777.953} C_VEL
LIN {X 0,Y 559.667,Z 613.974,A -85,B 0,C 180,E1 -2778.548,E2 -2778.548} C_VEL
LIN {X 0,Y 559.512,Z 625.175,A -85,B 0,C 180,E1 -2779.231,E2 -2779.231} C_VEL
LIN {X 0,Y 559.364,Z 633.767,A -85,B 0,C 180,E1 -2779.869,E2 -2779.869} C_VEL
LIN {X 0,Y 559.24,Z 641.997,A -85,B 0,C 180,E1 -2780.597,E2 -2780.597} C_VEL
LIN {X 0,Y 559.126,Z 650.54,A -85,B 0,C 180,E1 -2781.507,E2 -2781.507} C_VEL
LIN {X 0,Y 558.997,Z 657.621,A -85,B 0,C 180,E1 -2782.414,E2 -2782.414} C_VEL
LIN {X 0,Y 558.894,Z 664.602,A -85,B 0,C 180,E1 -2783.502,E2 -2783.502} C_VEL
LIN {X 0,Y 558.869,Z 670.18,A -85,B 0,C 180,E1 -2784.588,E2 -2784.588} C_VEL
LIN {X 0,Y 558.868,Z 674.54,A -85,B 0,C 180,E1 -2785.673,E2 -2785.673} C_VEL
LIN {X 0,Y 558.799,Z 678.666,A -85,B 0,C 180,E1 -2787.116,E2 -2787.116} C_VEL
LIN {X 0,Y 558.746,Z 680.14,A -85,B 0,C 180,E1 -2787.837,E2 -2787.837} C_VEL
LIN {X 0,Y 558.741,Z 681.739,A -85,B 0,C 180,E1 -2789.279,E2 -2789.279} C_VEL
LIN {X 0,Y 558.74,Z 681.996,A -85,B 0,C 180,E1 -2790,E2 -2790} C_VEL
LIN {X 0,Y 558.746,Z 681.224,A -85,B 0,C 180,E1 -2791.442,E2 -2791.442} C_VEL
LIN {X 0,Y 558.746,Z 680.279,A -85,B 0,C 180,E1 -2792.163,E2 -2792.163} C_VEL
LIN {X 0,Y 558.836,Z 677.062,A -85,B 0,C 180,E1 -2793.605,E2 -2793.605} C_VEL
LIN {X 0,Y 558.826,Z 673.503,A -85,B 0,C 180,E1 -2794.689,E2 -2794.689} C_VEL
LIN {X 0,Y 558.928,Z 668.853,A -85,B 0,C 180,E1 -2795.773,E2 -2795.773} C_VEL
LIN {X 0,Y 558.924,Z 663.185,A -85,B 0,C 180,E1 -2796.824,E2 -2796.824} C_VEL
LIN {X 0,Y 559.008,Z 656.962,A -85,B 0,C 180,E1 -2797.767,E2 -2797.767} C_VEL
LIN {X 0,Y 559.101,Z 649.754,A -85,B 0,C 180,E1 -2798.676,E2 -2798.676} C_VEL
LIN {X 0,Y 559.239,Z 641.062,A -85,B 0,C 180,E1 -2799.585,E2 -2799.585} C_VEL
LIN {X 0,Y 559.42,Z 630.343,A -85,B 0,C 180,E1 -2800.496,E2 -2800.496} C_VEL
LIN {X 0,Y 559.596,Z 618.902,A -85,B 0,C 180,E1 -2801.259,E2 -2801.259} C_VEL
LIN {X 0,Y 559.709,Z 610.071,A -85,B 0,C 180,E1 -2801.739,E2 -2801.739} C_VEL
LIN {X 0,Y 559.78,Z 598.82,A -85,B 0,C 180,E1 -2802.222,E2 -2802.222} C_VEL
LIN {X 0,Y 559.947,Z 587.803,A -85,B 0,C 180,E1 -2802.573,E2 -2802.573} C_VEL
LIN {X 0,Y 560.027,Z 577.518,A -85,B 0,C 180,E1 -2802.802,E2 -2802.802} C_VEL
LIN {X 0,Y 560.265,Z 476.021,A -85,B 0,C 180,E1 -2804.128,E2 -2804.128} C_VEL
LIN {X 0,Y 559.411,Z 469.602,A -85,B 0,C 180,E1 -2804.25,E2 -2804.25} C_VEL
LIN {X 0,Y 559.648,Z 447.968,A -85,B 0,C 180,E1 -2807.368,E2 -2807.368} C_VEL
LIN {X 0,Y 559.953,Z 427.318,A -85,B 0,C 180,E1 -2810.383,E2 -2810.383} C_VEL
LIN {X 0,Y 560.135,Z 410.051,A -85,B 0,C 180,E1 -2812.89,E2 -2812.89} C_VEL
LIN {X 0,Y 559.131,Z 403.842,A -85,B 0,C 180,E1 -2813.865,E2 -2813.865} C_VEL
LIN {X 0,Y 559.117,Z 403.836,A -85,B 0,C 180,E1 -2816.816,E2 -2816.816} C_VEL
LIN {X 0,Y 559.124,Z 403.84,A -85,B 0,C 180,E1 -2819.852,E2 -2819.852} C_VEL
LIN {X 0,Y 559.159,Z 403.83,A -85,B 0,C 180,E1 -2822.715,E2 -2822.715} C_VEL
LIN {X 0,Y 559.125,Z 403.842,A -85,B 0,C 180,E1 -2825.324,E2 -2825.324} C_VEL
LIN {X 0,Y 559.133,Z 403.833,A -85,B 0,C 180,E1 -2828.018,E2 -2828.018} C_VEL
LIN {X 0,Y 559.159,Z 403.831,A -85,B 0,C 180,E1 -2830.812,E2 -2830.812} C_VEL
LIN {X 0,Y 559.145,Z 403.831,A -85,B 0,C 180,E1 -2833.734,E2 -2833.734} C_VEL
LIN {X 0,Y 559.15,Z 403.837,A -85,B 0,C 180,E1 -2836.803,E2 -2836.803} C_VEL
LIN {X 0,Y 559.159,Z 403.834,A -85,B 0,C 180,E1 -2839.188,E2 -2839.188} C_VEL
LIN {X 0,Y 559.135,Z 403.832,A -85,B 0,C 180,E1 -2841.982,E2 -2841.982} C_VEL
LIN {X 0,Y 559.132,Z 403.84,A -85,B 0,C 180,E1 -2844.788,E2 -2844.788} C_VEL
LIN {X 0,Y 559.158,Z 403.83,A -85,B 0,C 180,E1 -2847.365,E2 -2847.365} C_VEL
LIN {X 0,Y 559.124,Z 403.838,A -85,B 0,C 180,E1 -2850.148,E2 -2850.148} C_VEL
LIN {X 0,Y 559.125,Z 403.834,A -85,B 0,C 180,E1 -2853.183,E2 -2853.183} C_VEL
LIN {X 0,Y 559.143,Z 403.84,A -85,B 0,C 180,E1 -2856.185,E2 -2856.185} C_VEL
LIN {X 0,Y 559.195,Z 404.223,A -85,B 0,C 180,E1 -2856.285,E2 -2856.285} C_VEL
LIN {X 0,Y 560.163,Z 409.625,A -85,B 0,C 180,E1 -2857.111,E2 -2857.111} C_VEL
LIN {X 0,Y 559.946,Z 429.329,A -85,B 0,C 180,E1 -2860,E2 -2860} C_VEL
LIN {X 0,Y 559.626,Z 449.346,A -85,B 0,C 180,E1 -2862.921,E2 -2862.921} C_VEL
LIN {X 0,Y 559.394,Z 469.622,A -85,B 0,C 180,E1 -2865.842,E2 -2865.842} C_VEL
LIN {X 0,Y 560.248,Z 475.601,A -85,B 0,C 180,E1 -2865.957,E2 -2865.957} C_VEL
LIN {X 0,Y 560.009,Z 577.683,A -85,B 0,C 180,E1 -2867.29,E2 -2867.29} C_VEL
LIN {X 0,Y 559.903,Z 589.677,A -85,B 0,C 180,E1 -2867.564,E2 -2867.564} C_VEL
LIN {X 0,Y 559.769,Z 603.376,A -85,B 0,C 180,E1 -2868.044,E2 -2868.044} C_VEL
LIN {X 0,Y 559.663,Z 614.355,A -85,B 0,C 180,E1 -2868.573,E2 -2868.573} C_VEL
LIN {X 0,Y 559.521,Z 623.81,A -85,B 0,C 180,E1 -2869.14,E2 -2869.14} C_VEL
LIN {X 0,Y 559.388,Z 632.615,A -85,B 0,C 180,E1 -2869.778,E2 -2869.778} C_VEL
LIN {X 0,Y 559.237,Z 642.014,A -85,B 0,C 180,E1 -2870.597,E2 -2870.597} C_VEL
LIN {X 0,Y 559.118,Z 650.61,A -85,B 0,C 180,E1 -2871.507,E2 -2871.507} C_VEL
LIN {X 0,Y 558.989,Z 658.938,A -85,B 0,C 180,E1 -2872.596,E2 -2872.596} C_VEL
LIN {X 0,Y 558.894,Z 664.614,A -85,B 0,C 180,E1 -2873.502,E2 -2873.502} C_VEL
LIN {X 0,Y 558.868,Z 670.146,A -85,B 0,C 180,E1 -2874.588,E2 -2874.588} C_VEL
LIN {X 0,Y 558.868,Z 674.485,A -85,B 0,C 180,E1 -2875.673,E2 -2875.673} C_VEL
LIN {X 0,Y 558.836,Z 676.842,A -85,B 0,C 180,E1 -2876.395,E2 -2876.395} C_VEL
LIN {X 0,Y 558.799,Z 678.675,A -85,B 0,C 180,E1 -2877.116,E2 -2877.116} C_VEL
LIN {X 0,Y 558.745,Z 681.144,A -85,B 0,C 180,E1 -2878.558,E2 -2878.558} C_VEL
LIN {X 0,Y 558.741,Z 681.753,A -85,B 0,C 180,E1 -2879.279,E2 -2879.279} C_VEL
LIN {X 0,Y 558.741,Z 681.809,A -85,B 0,C 180,E1 -2880.721,E2 -2880.721} C_VEL
LIN {X 0,Y 558.746,Z 681.241,A -85,B 0,C 180,E1 -2881.441,E2 -2881.441} C_VEL
LIN {X 0,Y 558.8,Z 678.893,A -85,B 0,C 180,E1 -2882.884,E2 -2882.884} C_VEL
LIN {X 0,Y 558.844,Z 676.016,A -85,B 0,C 180,E1 -2883.966,E2 -2883.966} C_VEL
LIN {X 0,Y 558.798,Z 672.104,A -85,B 0,C 180,E1 -2885.051,E2 -2885.051} C_VEL
LIN {X 0,Y 558.913,Z 667.048,A -85,B 0,C 180,E1 -2886.136,E2 -2886.136} C_VEL
LIN {X 0,Y 558.975,Z 660.7,A -85,B 0,C 180,E1 -2887.223,E2 -2887.223} C_VEL
LIN {X 0,Y 559.073,Z 652.845,A -85,B 0,C 180,E1 -2888.312,E2 -2888.312} C_VEL
LIN {X 0,Y 559.224,Z 642.966,A -85,B 0,C 180,E1 -2889.403,E2 -2889.403} C_VEL
LIN {X 0,Y 559.404,Z 633.749,A -85,B 0,C 180,E1 -2890.222,E2 -2890.222} C_VEL
LIN {X 0,Y 559.509,Z 623.968,A -85,B 0,C 180,E1 -2890.94,E2 -2890.94} C_VEL
LIN {X 0,Y 559.687,Z 613.021,A -85,B 0,C 180,E1 -2891.59,E2 -2891.59} C_VEL
LIN {X 0,Y 559.793,Z 599.917,A -85,B 0,C 180,E1 -2892.185,E2 -2892.185} C_VEL
LIN {X 0,Y 559.975,Z 587.836,A -85,B 0,C 180,E1 -2892.572,E2 -2892.572} C_VEL
LIN {X 0,Y 560.027,Z 577.561,A -85,B 0,C 180,E1 -2892.802,E2 -2892.802} C_VEL
LIN {X 0,Y 560.205,Z 475.404,A -85,B 0,C 180,E1 -2894.137,E2 -2894.137} C_VEL
LIN {X 0,Y 559.39,Z 469.603,A -85,B 0,C 180,E1 -2894.251,E2 -2894.251} C_VEL
LIN {X 0,Y 559.626,Z 449.982,A -85,B 0,C 180,E1 -2897.076,E2 -2897.076} C_VEL
LIN {X 0,Y 559.974,Z 428.64,A -85,B 0,C 180,E1 -2900.19,E2 -2900.19} C_VEL
LIN {X 0,Y 560.056,Z 409.596,A -85,B 0,C 180,E1 -2902.893,E2 -2902.893} C_VEL
LIN {X 0,Y 559.134,Z 403.841,A -85,B 0,C 180,E1 -2903.766,E2 -2903.766} C_VEL
LIN {X 0,Y 559.149,Z 403.836,A -85,B 0,C 180,E1 -2906.099,E2 -2906.099} C_VEL
LIN {X 0,Y 559.116,Z 403.836,A -85,B 0,C 180,E1 -2908.532,E2 -2908.532} C_VEL
LIN {X 0,Y 559.143,Z 403.838,A -85,B 0,C 180,E1 -2911.272,E2 -2911.272} C_VEL
LIN {X 0,Y 559.168,Z 403.831,A -85,B 0,C 180,E1 -2913.949,E2 -2913.949} C_VEL
LIN {X 0,Y 559.134,Z 403.838,A -85,B 0,C 180,E1 -2917.109,E2 -2917.109} C_VEL
LIN {X 0,Y 559.163,Z 403.829,A -85,B 0,C 180,E1 -2919.942,E2 -2919.942} C_VEL
LIN {X 0,Y 559.161,Z 403.833,A -85,B 0,C 180,E1 -2922.744,E2 -2922.744} C_VEL
LIN {X 0,Y 559.156,Z 403.83,A -85,B 0,C 180,E1 -2925.761,E2 -2925.761} C_VEL
LIN {X 0,Y 559.166,Z 403.83,A -85,B 0,C 180,E1 -2928.23,E2 -2928.23} C_VEL
LIN {X 0,Y 559.176,Z 403.83,A -85,B 0,C 180,E1 -2931.192,E2 -2931.192} C_VEL
LIN {X 0,Y 559.124,Z 403.834,A -85,B 0,C 180,E1 -2933.788,E2 -2933.788} C_VEL
LIN {X 0,Y 559.165,Z 403.836,A -85,B 0,C 180,E1 -2936.425,E2 -2936.425} C_VEL
LIN {X 0,Y 559.151,Z 403.833,A -85,B 0,C 180,E1 -2938.98,E2 -2938.98} C_VEL
LIN {X 0,Y 559.118,Z 403.837,A -85,B 0,C 180,E1 -2941.629,E2 -2941.629} C_VEL
LIN {X 0,Y 559.161,Z 403.885,A -85,B 0,C 180,E1 -2943.877,E2 -2943.877} C_VEL
LIN {X 0,Y 560.669,Z 411.946,A -85,B 0,C 180,E1 -2944.972,E2 -2944.972} C_VEL
LIN {X 0,Y 560.401,Z 433.721,A -85,B 0,C 180,E1 -2947.705,E2 -2947.705} C_VEL
LIN {X 0,Y 560.137,Z 452.163,A -85,B 0,C 180,E1 -2950.007,E2 -2950.007} C_VEL
LIN {X 0,Y 559.773,Z 476.58,A -85,B 0,C 180,E1 -2953.069,E2 -2953.069} C_VEL
LIN {X 0,Y 559.479,Z 498.64,A -85,B 0,C 180,E1 -2955.798,E2 -2955.798} C_VEL
LIN {X 0,Y 560.27,Z 505.502,A -85,B 0,C 180,E1 -2955.911,E2 -2955.911} C_VEL
LIN {X 0,Y 560.031,Z 607.943,A -85,B 0,C 180,E1 -2957.245,E2 -2957.245} C_VEL
LIN {X 0,Y 559.904,Z 621.216,A -85,B 0,C 180,E1 -2957.564,E2 -2957.564} C_VEL
LIN {X 0,Y 559.772,Z 632.918,A -85,B 0,C 180,E1 -2957.98,E2 -2957.98} C_VEL
LIN {X 0,Y 559.669,Z 644.808,A -85,B 0,C 180,E1 -2958.547,E2 -2958.547} C_VEL
LIN {X 0,Y 559.516,Z 655.906,A -85,B 0,C 180,E1 -2959.231,E2 -2959.231} C_VEL
LIN {X 0,Y 559.315,Z 666.539,A -85,B 0,C 180,E1 -2960.051,E2 -2960.051} C_VEL
LIN {X 0,Y 559.162,Z 676.112,A -85,B 0,C 180,E1 -2960.961,E2 -2960.961} C_VEL
LIN {X 0,Y 559.05,Z 683.96,A -85,B 0,C 180,E1 -2961.87,E2 -2961.87} C_VEL
LIN {X 0,Y 558.944,Z 691.622,A -85,B 0,C 180,E1 -2962.958,E2 -2962.958} C_VEL
LIN {X 0,Y 558.935,Z 698.68,A -85,B 0,C 180,E1 -2964.227,E2 -2964.227} C_VEL
LIN {X 0,Y 558.826,Z 703.372,A -85,B 0,C 180,E1 -2965.311,E2 -2965.311} C_VEL
LIN {X 0,Y 558.836,Z 706.958,A -85,B 0,C 180,E1 -2966.395,E2 -2966.395} C_VEL
LIN {X 0,Y 558.799,Z 708.808,A -85,B 0,C 180,E1 -2967.116,E2 -2967.116} C_VEL
LIN {X 0,Y 558.745,Z 711.185,A -85,B 0,C 180,E1 -2968.558,E2 -2968.558} C_VEL
LIN {X 0,Y 558.74,Z 712,A -85,B 0,C 180,E1 -2970,E2 -2970} C_VEL
LIN {X 0,Y 558.745,Z 711.186,A -85,B 0,C 180,E1 -2971.442,E2 -2971.442} C_VEL
LIN {X 0,Y 558.799,Z 708.81,A -85,B 0,C 180,E1 -2972.884,E2 -2972.884} C_VEL
LIN {X 0,Y 558.844,Z 705.896,A -85,B 0,C 180,E1 -2973.966,E2 -2973.966} C_VEL
LIN {X 0,Y 558.798,Z 701.949,A -85,B 0,C 180,E1 -2975.051,E2 -2975.051} C_VEL
LIN {X 0,Y 558.921,Z 696.867,A -85,B 0,C 180,E1 -2976.136,E2 -2976.136} C_VEL
LIN {X 0,Y 558.977,Z 690.468,A -85,B 0,C 180,E1 -2977.223,E2 -2977.223} C_VEL
LIN {X 0,Y 559.099,Z 682.477,A -85,B 0,C 180,E1 -2978.312,E2 -2978.312} C_VEL
LIN {X 0,Y 559.185,Z 674.334,A -85,B 0,C 180,E1 -2979.221,E2 -2979.221} C_VEL
LIN {X 0,Y 559.355,Z 664.399,A -85,B 0,C 180,E1 -2980.131,E2 -2980.131} C_VEL
LIN {X 0,Y 559.534,Z 653.404,A -85,B 0,C 180,E1 -2980.937,E2 -2980.937} C_VEL
LIN {X 0,Y 559.672,Z 641.459,A -85,B 0,C 180,E1 -2981.628,E2 -2981.628} C_VEL
LIN {X 0,Y 559.817,Z 628.766,A -85,B 0,C 180,E1 -2982.185,E2 -2982.185} C_VEL
LIN {X 0,Y 559.967,Z 615.344,A -85,B 0,C 180,E1 -2982.596,E2 -2982.596} C_VEL
LIN {X 0,Y 560.066,Z 602.079,A -85,B 0,C 180,E1 -2982.847,E2 -2982.847} C_VEL
LIN {X 0,Y 560.174,Z 503.714,A -85,B 0,C 180,E1 -2984.115,E2 -2984.115} C_VEL
LIN {X 0,Y 559.493,Z 498.452,A -85,B 0,C 180,E1 -2984.225,E2 -2984.225} C_VEL
LIN {X 0,Y 559.83,Z 472.587,A -85,B 0,C 180,E1 -2987.428,E2 -2987.428} C_VEL
LIN {X 0,Y 560.209,Z 449.153,A -85,B 0,C 180,E1 -2990.373,E2 -2990.373} C_VEL
LIN {X 0,Y 560.398,Z 427.159,A -85,B 0,C 180,E1 -2993.073,E2 -2993.073} C_VEL
LIN {X 0,Y 560.506,Z 411.208,A -85,B 0,C 180,E1 -2995.036,E2 -2995.036} C_VEL
LIN {X 0,Y 559.181,Z 403.835,A -85,B 0,C 180,E1 -2996,E2 -2996} C_VEL
LIN {X 0,Y 559.116,Z 403.837,A -85,B 0,C 180,E1 -2998.532,E2 -2998.532} C_VEL
LIN {X 0,Y 559.143,Z 403.837,A -85,B 0,C 180,E1 -3001.272,E2 -3001.272} C_VEL
LIN {X 0,Y 559.167,Z 403.832,A -85,B 0,C 180,E1 -3003.949,E2 -3003.949} C_VEL
LIN {X 0,Y 559.132,Z 403.837,A -85,B 0,C 180,E1 -3007.109,E2 -3007.109} C_VEL
LIN {X 0,Y 559.162,Z 403.831,A -85,B 0,C 180,E1 -3009.942,E2 -3009.942} C_VEL
LIN {X 0,Y 559.157,Z 403.831,A -85,B 0,C 180,E1 -3012.744,E2 -3012.744} C_VEL
LIN {X 0,Y 559.155,Z 403.832,A -85,B 0,C 180,E1 -3015.761,E2 -3015.761} C_VEL
LIN {X 0,Y 559.166,Z 403.828,A -85,B 0,C 180,E1 -3018.23,E2 -3018.23} C_VEL
LIN {X 0,Y 559.178,Z 403.835,A -85,B 0,C 180,E1 -3021.192,E2 -3021.192} C_VEL
LIN {X 0,Y 559.142,Z 403.832,A -85,B 0,C 180,E1 -3023.789,E2 -3023.789} C_VEL
LIN {X 0,Y 559.166,Z 403.83,A -85,B 0,C 180,E1 -3026.425,E2 -3026.425} C_VEL
LIN {X 0,Y 559.158,Z 403.838,A -85,B 0,C 180,E1 -3028.981,E2 -3028.981} C_VEL
LIN {X 0,Y 559.149,Z 403.831,A -85,B 0,C 180,E1 -3031.623,E2 -3031.623} C_VEL
LIN {X 0,Y 559.177,Z 403.828,A -85,B 0,C 180,E1 -3033.903,E2 -3033.903} C_VEL
LIN {X 0,Y 559.146,Z 403.84,A -85,B 0,C 180,E1 -3036.571,E2 -3036.571} C_VEL
LIN {X 0,Y 559.177,Z 403.828,A -85,B 0,C 180,E1 -3039.395,E2 -3039.395} C_VEL
LIN {X 0,Y 559.134,Z 403.834,A -85,B 0,C 180,E1 -3041.685,E2 -3041.685} C_VEL
LIN {X 0,Y 559.146,Z 403.834,A -85,B 0,C 180,E1 -3043.947,E2 -3043.947} C_VEL
LIN {X 0,Y 559.143,Z 403.837,A -85,B 0,C 180,E1 -3045.905,E2 -3045.905} C_VEL
LIN {X 0,Y 560.291,Z 409.977,A -85,B 0,C 180,E1 -3046.014,E2 -3046.014} C_VEL
LIN {X 0,Y 560.048,Z 507.684,A -85,B 0,C 180,E1 -3047.291,E2 -3047.291} C_VEL
LIN {X 0,Y 559.933,Z 520.564,A -85,B 0,C 180,E1 -3047.588,E2 -3047.588} C_VEL
LIN {X 0,Y 559.781,Z 533.326,A -85,B 0,C 180,E1 -3048.045,E2 -3048.045} C_VEL
LIN {X 0,Y 559.667,Z 543.874,A -85,B 0,C 180,E1 -3048.548,E2 -3048.548} C_VEL
LIN {X 0,Y 559.532,Z 553.8,A -85,B 0,C 180,E1 -3049.14,E2 -3049.14} C_VEL
LIN {X 0,Y 559.364,Z 563.792,A -85,B 0,C 180,E1 -3049.869,E2 -3049.869} C_VEL
LIN {X 0,Y 559.21,Z 573.909,A -85,B 0,C 180,E1 -3050.779,E2 -3050.779} C_VEL
LIN {X 0,Y 559.082,Z 582.094,A -85,B 0,C 180,E1 -3051.688,E2 -3051.688} C_VEL
LIN {X 0,Y 558.974,Z 588.895,A -85,B 0,C 180,E1 -3052.596,E2 -3052.596} C_VEL
LIN {X 0,Y 558.889,Z 595.375,A -85,B 0,C 180,E1 -3053.645,E2 -3053.645} C_VEL
LIN {X 0,Y 558.869,Z 600.129,A -85,B 0,C 180,E1 -3054.588,E2 -3054.588} C_VEL
LIN {X 0,Y 558.869,Z 604.506,A -85,B 0,C 180,E1 -3055.673,E2 -3055.673} C_VEL
LIN {X 0,Y 558.799,Z 608.695,A -85,B 0,C 180,E1 -3057.116,E2 -3057.116} C_VEL
LIN {X 0,Y 558.746,Z 610.129,A -85,B 0,C 180,E1 -3057.837,E2 -3057.837} C_VEL
LIN {X 0,Y 558.741,Z 611.746,A -85,B 0,C 180,E1 -3059.279,E2 -3059.279} C_VEL
LIN {X 0,Y 558.74,Z 611.996,A -85,B 0,C 180,E1 -3060,E2 -3060} C_VEL
LIN {X 0,Y 558.746,Z 611.21,A -85,B 0,C 180,E1 -3061.442,E2 -3061.442} C_VEL
LIN {X 0,Y 558.746,Z 610.283,A -85,B 0,C 180,E1 -3062.163,E2 -3062.163} C_VEL
LIN {X 0,Y 558.8,Z 608.871,A -85,B 0,C 180,E1 -3062.884,E2 -3062.884} C_VEL
LIN {X 0,Y 558.869,Z 604.838,A -85,B 0,C 180,E1 -3064.327,E2 -3064.327} C_VEL
LIN {X 0,Y 558.868,Z 600.547,A -85,B 0,C 180,E1 -3065.412,E2 -3065.412} C_VEL
LIN {X 0,Y 558.894,Z 595.074,A -85,B 0,C 180,E1 -3066.498,E2 -3066.498} C_VEL
LIN {X 0,Y 558.971,Z 589.495,A -85,B 0,C 180,E1 -3067.405,E2 -3067.405} C_VEL
LIN {X 0,Y 559.073,Z 582.803,A -85,B 0,C 180,E1 -3068.312,E2 -3068.312} C_VEL
LIN {X 0,Y 559.195,Z 574.77,A -85,B 0,C 180,E1 -3069.221,E2 -3069.221} C_VEL
LIN {X 0,Y 559.404,Z 563.78,A -85,B 0,C 180,E1 -3070.222,E2 -3070.222} C_VEL
LIN {X 0,Y 559.509,Z 553.951,A -85,B 0,C 180,E1 -3070.94,E2 -3070.94} C_VEL
LIN {X 0,Y 559.657,Z 544.688,A -85,B 0,C 180,E1 -3071.497,E2 -3071.497} C_VEL
LIN {X 0,Y 559.747,Z 534.317,A -85,B 0,C 180,E1 -3072.002,E2 -3072.002} C_VEL
LIN {X 0,Y 559.896,Z 523.349,A -85,B 0,C 180,E1 -3072.413,E2 -3072.413} C_VEL
LIN {X 0,Y 560.035,Z 508.919,A -85,B 0,C 180,E1 -3072.778,E2 -3072.778} C_VEL
LIN {X 0,Y 560.181,Z 473.382,A -85,B 0,C 180,E1 -3073.259,E2 -3073.259} C_VEL
LIN {X 0,Y 560.221,Z 409.201,A -85,B 0,C 180,E1 -3074.088,E2 -3074.088} C_VEL
LIN {X 0,Y 559.168,Z 403.832,A -85,B 0,C 180,E1 -3074.187,E2 -3074.187} C_VEL
LIN {X 0,Y 559.146,Z 403.833,A -85,B 0,C 180,E1 -3076.968,E2 -3076.968} C_VEL
LIN {X 0,Y 558.498,Z 403.921,A -85,B 0,C 180,E1 -3077.569,E2 -3077.569} C_VEL
LIN {X 0,Y 555.674,Z 404.272,A -85,B 0,C 180,E1 -3078.544,E2 -3078.544} C_VEL
LIN {X 0,Y 553.268,Z 404.571,A -85,B 0,C 180,E1 -3079.329,E2 -3079.329} C_VEL
LIN {X 0,Y 552.219,Z 404.698,A -85,B 0,C 180,E1 -3079.935,E2 -3079.935} C_VEL
LIN {X 0,Y 552.125,Z 404.708,A -85,B 0,C 180,E1 -3080.14,E2 -3080.14} C_VEL
LIN {X 0,Y 552.091,Z 404.709,A -85,B 0,C 180,E1 -3082.451,E2 -3082.451} C_VEL
LIN {X 0,Y 552.089,Z 404.719,A -85,B 0,C 180,E1 -3085.335,E2 -3085.335} C_VEL
LIN {X 0,Y 552.092,Z 404.708,A -85,B 0,C 180,E1 -3088.099,E2 -3088.099} C_VEL
LIN {X 0,Y 552.105,Z 404.709,A -85,B 0,C 180,E1 -3090.609,E2 -3090.609} C_VEL
LIN {X 0,Y 552.119,Z 404.709,A -85,B 0,C 180,E1 -3093.186,E2 -3093.186} C_VEL
LIN {X 0,Y 552.089,Z 404.71,A -85,B 0,C 180,E1 -3095.844,E2 -3095.844} C_VEL
LIN {X 0,Y 552.121,Z 404.71,A -85,B 0,C 180,E1 -3098.589,E2 -3098.589} C_VEL
LIN {X 0,Y 552.124,Z 404.707,A -85,B 0,C 180,E1 -3101.446,E2 -3101.446} C_VEL
LIN {X 0,Y 552.097,Z 404.714,A -85,B 0,C 180,E1 -3104.532,E2 -3104.532} C_VEL
LIN {X 0,Y 552.133,Z 404.704,A -85,B 0,C 180,E1 -3107.585,E2 -3107.585} C_VEL
LIN {X 0,Y 552.131,Z 404.709,A -85,B 0,C 180,E1 -3110.473,E2 -3110.473} C_VEL
LIN {X 0,Y 552.101,Z 404.708,A -85,B 0,C 180,E1 -3113.318,E2 -3113.318} C_VEL
LIN {X 0,Y 552.128,Z 404.706,A -85,B 0,C 180,E1 -3115.939,E2 -3115.939} C_VEL
LIN {X 0,Y 552.123,Z 404.715,A -85,B 0,C 180,E1 -3118.541,E2 -3118.541} C_VEL
LIN {X 0,Y 552.086,Z 404.712,A -85,B 0,C 180,E1 -3121.446,E2 -3121.446} C_VEL
LIN {X 0,Y 552.082,Z 404.72,A -85,B 0,C 180,E1 -3124.353,E2 -3124.353} C_VEL
LIN {X 0,Y 552.126,Z 404.883,A -85,B 0,C 180,E1 -3126.149,E2 -3126.149} C_VEL
LIN {X 0,Y 553.215,Z 411.784,A -85,B 0,C 180,E1 -3127.203,E2 -3127.203} C_VEL
LIN {X 0,Y 552.958,Z 431.895,A -85,B 0,C 180,E1 -3130.141,E2 -3130.141} C_VEL
LIN {X 0,Y 552.62,Z 451.346,A -85,B 0,C 180,E1 -3132.992,E2 -3132.992} C_VEL
LIN {X 0,Y 552.407,Z 469.868,A -85,B 0,C 180,E1 -3135.677,E2 -3135.677} C_VEL
LIN {X 0,Y 553.367,Z 477.761,A -85,B 0,C 180,E1 -3135.806,E2 -3135.806} C_VEL
LIN {X 0,Y 553.098,Z 577.622,A -85,B 0,C 180,E1 -3137.129,E2 -3137.129} C_VEL
LIN {X 0,Y 553.002,Z 587.87,A -85,B 0,C 180,E1 -3137.36,E2 -3137.36} C_VEL
LIN {X 0,Y 552.863,Z 598.616,A -85,B 0,C 180,E1 -3137.706,E2 -3137.706} C_VEL
LIN {X 0,Y 552.801,Z 607.396,A -85,B 0,C 180,E1 -3138.077,E2 -3138.077} C_VEL
LIN {X 0,Y 552.654,Z 616.962,A -85,B 0,C 180,E1 -3138.576,E2 -3138.576} C_VEL
LIN {X 0,Y 552.507,Z 626.479,A -85,B 0,C 180,E1 -3139.186,E2 -3139.186} C_VEL
LIN {X 0,Y 552.312,Z 634.856,A -85,B 0,C 180,E1 -3139.831,E2 -3139.831} C_VEL
LIN {X 0,Y 552.205,Z 641.991,A -85,B 0,C 180,E1 -3140.476,E2 -3140.476} C_VEL
LIN {X 0,Y 552.094,Z 650.534,A -85,B 0,C 180,E1 -3141.398,E2 -3141.398} C_VEL
LIN {X 0,Y 551.95,Z 657.616,A -85,B 0,C 180,E1 -3142.317,E2 -3142.317} C_VEL
LIN {X 0,Y 551.843,Z 664.597,A -85,B 0,C 180,E1 -3143.418,E2 -3143.418} C_VEL
LIN {X 0,Y 551.804,Z 670.181,A -85,B 0,C 180,E1 -3144.519,E2 -3144.519} C_VEL
LIN {X 0,Y 551.764,Z 674.544,A -85,B 0,C 180,E1 -3145.617,E2 -3145.617} C_VEL
LIN {X 0,Y 551.723,Z 678.66,A -85,B 0,C 180,E1 -3147.079,E2 -3147.079} C_VEL
LIN {X 0,Y 551.656,Z 680.141,A -85,B 0,C 180,E1 -3147.81,E2 -3147.81} C_VEL
LIN {X 0,Y 551.642,Z 681.732,A -85,B 0,C 180,E1 -3149.27,E2 -3149.27} C_VEL
LIN {X 0,Y 551.641,Z 681.996,A -85,B 0,C 180,E1 -3150,E2 -3150} C_VEL
LIN {X 0,Y 551.645,Z 681.216,A -85,B 0,C 180,E1 -3151.46,E2 -3151.46} C_VEL
LIN {X 0,Y 551.657,Z 680.28,A -85,B 0,C 180,E1 -3152.19,E2 -3152.19} C_VEL
LIN {X 0,Y 551.751,Z 677.054,A -85,B 0,C 180,E1 -3153.652,E2 -3153.652} C_VEL
LIN {X 0,Y 551.725,Z 673.494,A -85,B 0,C 180,E1 -3154.749,E2 -3154.749} C_VEL
LIN {X 0,Y 551.859,Z 668.842,A -85,B 0,C 180,E1 -3155.848,E2 -3155.848} C_VEL
LIN {X 0,Y 551.836,Z 664.042,A -85,B 0,C 180,E1 -3156.765,E2 -3156.765} C_VEL
LIN {X 0,Y 551.949,Z 658.254,A -85,B 0,C 180,E1 -3157.683,E2 -3157.683} C_VEL
LIN {X 0,Y 552.065,Z 651.293,A -85,B 0,C 180,E1 -3158.603,E2 -3158.603} C_VEL
LIN {X 0,Y 552.152,Z 644.734,A -85,B 0,C 180,E1 -3159.34,E2 -3159.34} C_VEL
LIN {X 0,Y 552.288,Z 635.921,A -85,B 0,C 180,E1 -3160.17,E2 -3160.17} C_VEL
LIN {X 0,Y 552.479,Z 627.75,A -85,B 0,C 180,E1 -3160.815,E2 -3160.815} C_VEL
LIN {X 0,Y 552.637,Z 618.543,A -85,B 0,C 180,E1 -3161.422,E2 -3161.422} C_VEL
LIN {X 0,Y 552.75,Z 609.297,A -85,B 0,C 180,E1 -3161.924,E2 -3161.924} C_VEL
LIN {X 0,Y 552.831,Z 599.79,A -85,B 0,C 180,E1 -3162.341,E2 -3162.341} C_VEL
LIN {X 0,Y 553.025,Z 588.609,A -85,B 0,C 180,E1 -3162.71,E2 -3162.71} C_VEL
LIN {X 0,Y 553.089,Z 578.753,A -85,B 0,C 180,E1 -3162.942,E2 -3162.942} C_VEL
LIN {X 0,Y 553.231,Z 550.495,A -85,B 0,C 180,E1 -3163.335,E2 -3163.335} C_VEL
LIN {X 0,Y 553.297,Z 475.839,A -85,B 0,C 180,E1 -3164.311,E2 -3164.311} C_VEL
LIN {X 0,Y 552.405,Z 469.665,A -85,B 0,C 180,E1 -3164.425,E2 -3164.425} C_VEL
LIN {X 0,Y 552.683,Z 448.603,A -85,B 0,C 180,E1 -3167.5,E2 -3167.5} C_VEL
LIN {X 0,Y 552.994,Z 427.095,A -85,B 0,C 180,E1 -3170.651,E2 -3170.651} C_VEL
LIN {X 0,Y 553.178,Z 411.058,A -85,B 0,C 180,E1 -3172.996,E2 -3172.996} C_VEL
LIN {X 0,Y 552.093,Z 404.718,A -85,B 0,C 180,E1 -3173.979,E2 -3173.979} C_VEL
LIN {X 0,Y 552.08,Z 404.714,A -85,B 0,C 180,E1 -3176.987,E2 -3176.987} C_VEL
LIN {X 0,Y 552.099,Z 404.712,A -85,B 0,C 180,E1 -3180.047,E2 -3180.047} C_VEL
LIN {X 0,Y 552.117,Z 404.708,A -85,B 0,C 180,E1 -3182.846,E2 -3182.846} C_VEL
LIN {X 0,Y 552.073,Z 404.721,A -85,B 0,C 180,E1 -3185.439,E2 -3185.439} C_VEL
LIN {X 0,Y 552.096,Z 404.711,A -85,B 0,C 180,E1 -3187.885,E2 -3187.885} C_VEL
LIN {X 0,Y 552.112,Z 404.706,A -85,B 0,C 180,E1 -3190.481,E2 -3190.481} C_VEL
LIN {X 0,Y 552.123,Z 404.708,A -85,B 0,C 180,E1 -3193.485,E2 -3193.485} C_VEL
LIN {X 0,Y 552.11,Z 404.711,A -85,B 0,C 180,E1 -3196.576,E2 -3196.576} C_VEL
LIN {X 0,Y 552.113,Z 404.708,A -85,B 0,C 180,E1 -3199.519,E2 -3199.519} C_VEL
LIN {X 0,Y 552.093,Z 404.712,A -85,B 0,C 180,E1 -3202.336,E2 -3202.336} C_VEL
LIN {X 0,Y 552.085,Z 404.714,A -85,B 0,C 180,E1 -3205.051,E2 -3205.051} C_VEL
LIN {X 0,Y 552.117,Z 404.706,A -85,B 0,C 180,E1 -3207.681,E2 -3207.681} C_VEL
LIN {X 0,Y 552.089,Z 404.716,A -85,B 0,C 180,E1 -3210.234,E2 -3210.234} C_VEL
LIN {X 0,Y 552.095,Z 404.711,A -85,B 0,C 180,E1 -3213.01,E2 -3213.01} C_VEL
LIN {X 0,Y 552.117,Z 404.775,A -85,B 0,C 180,E1 -3216.1,E2 -3216.1} C_VEL
LIN {X 0,Y 553.27,Z 412.044,A -85,B 0,C 180,E1 -3217.205,E2 -3217.205} C_VEL
LIN {X 0,Y 552.954,Z 431.869,A -85,B 0,C 180,E1 -3220.142,E2 -3220.142} C_VEL
LIN {X 0,Y 552.648,Z 450.111,A -85,B 0,C 180,E1 -3222.811,E2 -3222.811} C_VEL
LIN {X 0,Y 552.425,Z 469.945,A -85,B 0,C 180,E1 -3225.678,E2 -3225.678} C_VEL
LIN {X 0,Y 553.369,Z 477.817,A -85,B 0,C 180,E1 -3225.807,E2 -3225.807} C_VEL
LIN {X 0,Y 553.098,Z 577.67,A -85,B 0,C 180,E1 -3227.129,E2 -3227.129} C_VEL
LIN {X 0,Y 552.969,Z 589.671,A -85,B 0,C 180,E1 -3227.405,E2 -3227.405} C_VEL
LIN {X 0,Y 552.818,Z 603.362,A -85,B 0,C 180,E1 -3227.891,E2 -3227.891} C_VEL
LIN {X 0,Y 552.652,Z 613.305,A -85,B 0,C 180,E1 -3228.368,E2 -3228.368} C_VEL
LIN {X 0,Y 552.534,Z 623.805,A -85,B 0,C 180,E1 -3229.001,E2 -3229.001} C_VEL
LIN {X 0,Y 552.378,Z 632.612,A -85,B 0,C 180,E1 -3229.647,E2 -3229.647} C_VEL
LIN {X 0,Y 552.244,Z 640.057,A -85,B 0,C 180,E1 -3230.292,E2 -3230.292} C_VEL
LIN {X 0,Y 552.124,Z 647.314,A -85,B 0,C 180,E1 -3231.029,E2 -3231.029} C_VEL
LIN {X 0,Y 551.985,Z 654.939,A -85,B 0,C 180,E1 -3231.949,E2 -3231.949} C_VEL
LIN {X 0,Y 551.888,Z 661.401,A -85,B 0,C 180,E1 -3232.886,E2 -3232.886} C_VEL
LIN {X 0,Y 551.839,Z 667.175,A -85,B 0,C 180,E1 -3233.901,E2 -3233.901} C_VEL
LIN {X 0,Y 551.739,Z 673.215,A -85,B 0,C 180,E1 -3235.251,E2 -3235.251} C_VEL
LIN {X 0,Y 551.75,Z 676.846,A -85,B 0,C 180,E1 -3236.348,E2 -3236.348} C_VEL
LIN {X 0,Y 551.723,Z 678.673,A -85,B 0,C 180,E1 -3237.079,E2 -3237.079} C_VEL
LIN {X 0,Y 551.645,Z 681.145,A -85,B 0,C 180,E1 -3238.54,E2 -3238.54} C_VEL
LIN {X 0,Y 551.642,Z 681.753,A -85,B 0,C 180,E1 -3239.27,E2 -3239.27} C_VEL
LIN {X 0,Y 551.641,Z 681.809,A -85,B 0,C 180,E1 -3240.73,E2 -3240.73} C_VEL
LIN {X 0,Y 551.646,Z 681.236,A -85,B 0,C 180,E1 -3241.46,E2 -3241.46} C_VEL
LIN {X 0,Y 551.724,Z 678.888,A -85,B 0,C 180,E1 -3242.921,E2 -3242.921} C_VEL
LIN {X 0,Y 551.764,Z 676.008,A -85,B 0,C 180,E1 -3244.017,E2 -3244.017} C_VEL
LIN {X 0,Y 551.723,Z 672.094,A -85,B 0,C 180,E1 -3245.116,E2 -3245.116} C_VEL
LIN {X 0,Y 551.84,Z 667.646,A -85,B 0,C 180,E1 -3246.099,E2 -3246.099} C_VEL
LIN {X 0,Y 551.886,Z 661.855,A -85,B 0,C 180,E1 -3247.132,E2 -3247.132} C_VEL
LIN {X 0,Y 551.983,Z 655.62,A -85,B 0,C 180,E1 -3248.051,E2 -3248.051} C_VEL
LIN {X 0,Y 552.102,Z 648.121,A -85,B 0,C 180,E1 -3248.971,E2 -3248.971} C_VEL
LIN {X 0,Y 552.226,Z 641.006,A -85,B 0,C 180,E1 -3249.708,E2 -3249.708} C_VEL
LIN {X 0,Y 552.407,Z 632.581,A -85,B 0,C 180,E1 -3250.445,E2 -3250.445} C_VEL
LIN {X 0,Y 552.552,Z 622.91,A -85,B 0,C 180,E1 -3251.15,E2 -3251.15} C_VEL
LIN {X 0,Y 552.739,Z 611.291,A -85,B 0,C 180,E1 -3251.831,E2 -3251.831} C_VEL
LIN {X 0,Y 552.865,Z 598.583,A -85,B 0,C 180,E1 -3252.387,E2 -3252.387} C_VEL
LIN {X 0,Y 553.043,Z 587.785,A -85,B 0,C 180,E1 -3252.733,E2 -3252.733} C_VEL
LIN {X 0,Y 553.117,Z 577.479,A -85,B 0,C 180,E1 -3252.964,E2 -3252.964} C_VEL
LIN {X 0,Y 553.297,Z 475.849,A -85,B 0,C 180,E1 -3254.311,E2 -3254.311} C_VEL
LIN {X 0,Y 552.398,Z 469.734,A -85,B 0,C 180,E1 -3254.416,E2 -3254.416} C_VEL
LIN {X 0,Y 552.673,Z 448.628,A -85,B 0,C 180,E1 -3257.497,E2 -3257.497} C_VEL
LIN {X 0,Y 552.97,Z 428.38,A -85,B 0,C 180,E1 -3260.458,E2 -3260.458} C_VEL
LIN {X 0,Y 553.108,Z 411.796,A -85,B 0,C 180,E1 -3262.802,E2 -3262.802} C_VEL
LIN {X 0,Y 552.379,Z 406.155,A -85,B 0,C 180,E1 -3263.642,E2 -3263.642} C_VEL
LIN {X 0,Y 552.112,Z 404.716,A -85,B 0,C 180,E1 -3263.884,E2 -3263.884} C_VEL
LIN {X 0,Y 552.08,Z 404.714,A -85,B 0,C 180,E1 -3266.987,E2 -3266.987} C_VEL
LIN {X 0,Y 552.099,Z 404.714,A -85,B 0,C 180,E1 -3270.047,E2 -3270.047} C_VEL
LIN {X 0,Y 552.117,Z 404.709,A -85,B 0,C 180,E1 -3272.846,E2 -3272.846} C_VEL
LIN {X 0,Y 552.073,Z 404.721,A -85,B 0,C 180,E1 -3275.439,E2 -3275.439} C_VEL
LIN {X 0,Y 552.096,Z 404.711,A -85,B 0,C 180,E1 -3277.885,E2 -3277.885} C_VEL
LIN {X 0,Y 552.111,Z 404.708,A -85,B 0,C 180,E1 -3280.481,E2 -3280.481} C_VEL
LIN {X 0,Y 552.122,Z 404.71,A -85,B 0,C 180,E1 -3283.485,E2 -3283.485} C_VEL
LIN {X 0,Y 552.109,Z 404.712,A -85,B 0,C 180,E1 -3286.576,E2 -3286.576} C_VEL
LIN {X 0,Y 552.111,Z 404.708,A -85,B 0,C 180,E1 -3289.519,E2 -3289.519} C_VEL
LIN {X 0,Y 552.091,Z 404.713,A -85,B 0,C 180,E1 -3292.336,E2 -3292.336} C_VEL
LIN {X 0,Y 552.084,Z 404.714,A -85,B 0,C 180,E1 -3295.051,E2 -3295.051} C_VEL
LIN {X 0,Y 552.116,Z 404.707,A -85,B 0,C 180,E1 -3297.681,E2 -3297.681} C_VEL
LIN {X 0,Y 552.088,Z 404.717,A -85,B 0,C 180,E1 -3300.234,E2 -3300.234} C_VEL
LIN {X 0,Y 552.08,Z 404.716,A -85,B 0,C 180,E1 -3303.012,E2 -3303.012} C_VEL
LIN {X 0,Y 552.119,Z 404.745,A -85,B 0,C 180,E1 -3303.696,E2 -3303.696} C_VEL
LIN {X 0,Y 553.747,Z 413.015,A -85,B 0,C 180,E1 -3304.838,E2 -3304.838} C_VEL
LIN {X 0,Y 553.445,Z 434.75,A -85,B 0,C 180,E1 -3307.607,E2 -3307.607} C_VEL
LIN {X 0,Y 553.149,Z 455.493,A -85,B 0,C 180,E1 -3310.203,E2 -3310.203} C_VEL
LIN {X 0,Y 552.798,Z 477.754,A -85,B 0,C 180,E1 -3312.998,E2 -3312.998} C_VEL
LIN {X 0,Y 552.503,Z 498.64,A -85,B 0,C 180,E1 -3315.615,E2 -3315.615} C_VEL
LIN {X 0,Y 553.402,Z 506.112,A -85,B 0,C 180,E1 -3315.74,E2 -3315.74} C_VEL
LIN {X 0,Y 553.123,Z 607.943,A -85,B 0,C 180,E1 -3317.083,E2 -3317.083} C_VEL
LIN {X 0,Y 552.965,Z 621.215,A -85,B 0,C 180,E1 -3317.405,E2 -3317.405} C_VEL
LIN {X 0,Y 552.833,Z 633.368,A -85,B 0,C 180,E1 -3317.845,E2 -3317.845} C_VEL
LIN {X 0,Y 552.685,Z 645.712,A -85,B 0,C 180,E1 -3318.452,E2 -3318.452} C_VEL
LIN {X 0,Y 552.477,Z 657.196,A -85,B 0,C 180,E1 -3319.185,E2 -3319.185} C_VEL
LIN {X 0,Y 552.301,Z 667.603,A -85,B 0,C 180,E1 -3320.016,E2 -3320.016} C_VEL
LIN {X 0,Y 552.126,Z 676.112,A -85,B 0,C 180,E1 -3320.845,E2 -3320.845} C_VEL
LIN {X 0,Y 552.013,Z 683.96,A -85,B 0,C 180,E1 -3321.765,E2 -3321.765} C_VEL
LIN {X 0,Y 551.889,Z 691.621,A -85,B 0,C 180,E1 -3322.868,E2 -3322.868} C_VEL
LIN {X 0,Y 551.867,Z 698.68,A -85,B 0,C 180,E1 -3324.153,E2 -3324.153} C_VEL
LIN {X 0,Y 551.725,Z 703.372,A -85,B 0,C 180,E1 -3325.251,E2 -3325.251} C_VEL
LIN {X 0,Y 551.75,Z 706.958,A -85,B 0,C 180,E1 -3326.348,E2 -3326.348} C_VEL
LIN {X 0,Y 551.723,Z 708.807,A -85,B 0,C 180,E1 -3327.079,E2 -3327.079} C_VEL
LIN {X 0,Y 551.645,Z 711.184,A -85,B 0,C 180,E1 -3328.54,E2 -3328.54} C_VEL
LIN {X 0,Y 551.64,Z 712,A -85,B 0,C 180,E1 -3330,E2 -3330} C_VEL
LIN {X 0,Y 551.645,Z 711.185,A -85,B 0,C 180,E1 -3331.46,E2 -3331.46} C_VEL
LIN {X 0,Y 551.723,Z 708.81,A -85,B 0,C 180,E1 -3332.921,E2 -3332.921} C_VEL
LIN {X 0,Y 551.764,Z 705.895,A -85,B 0,C 180,E1 -3334.017,E2 -3334.017} C_VEL
LIN {X 0,Y 551.723,Z 701.948,A -85,B 0,C 180,E1 -3335.116,E2 -3335.116} C_VEL
LIN {X 0,Y 551.803,Z 696.188,A -85,B 0,C 180,E1 -3336.342,E2 -3336.342} C_VEL
LIN {X 0,Y 551.926,Z 689.236,A -85,B 0,C 180,E1 -3337.5,E2 -3337.5} C_VEL
LIN {X 0,Y 552.082,Z 680.991,A -85,B 0,C 180,E1 -3338.602,E2 -3338.602} C_VEL
LIN {X 0,Y 552.224,Z 672.539,A -85,B 0,C 180,E1 -3339.523,E2 -3339.523} C_VEL
LIN {X 0,Y 552.424,Z 662.094,A -85,B 0,C 180,E1 -3340.445,E2 -3340.445} C_VEL
LIN {X 0,Y 552.606,Z 651.298,A -85,B 0,C 180,E1 -3341.213,E2 -3341.213} C_VEL
LIN {X 0,Y 552.751,Z 640.405,A -85,B 0,C 180,E1 -3341.831,E2 -3341.831} C_VEL
LIN {X 0,Y 552.876,Z 628.762,A -85,B 0,C 180,E1 -3342.34,E2 -3342.34} C_VEL
LIN {X 0,Y 553.042,Z 615.343,A -85,B 0,C 180,E1 -3342.756,E2 -3342.756} C_VEL
LIN {X 0,Y 553.167,Z 602.079,A -85,B 0,C 180,E1 -3343.01,E2 -3343.01} C_VEL
LIN {X 0,Y 553.368,Z 504.954,A -85,B 0,C 180,E1 -3344.276,E2 -3344.276} C_VEL
LIN {X 0,Y 552.513,Z 498.64,A -85,B 0,C 180,E1 -3344.385,E2 -3344.385} C_VEL
LIN {X 0,Y 552.886,Z 473.275,A -85,B 0,C 180,E1 -3347.567,E2 -3347.567} C_VEL
LIN {X 0,Y 553.158,Z 453.209,A -85,B 0,C 180,E1 -3350.062,E2 -3350.062} C_VEL
LIN {X 0,Y 553.374,Z 434.229,A -85,B 0,C 180,E1 -3352.396,E2 -3352.396} C_VEL
LIN {X 0,Y 553.586,Z 413.522,A -85,B 0,C 180,E1 -3354.969,E2 -3354.969} C_VEL
LIN {X 0,Y 552.564,Z 406.993,A -85,B 0,C 180,E1 -3355.825,E2 -3355.825} C_VEL
LIN {X 0,Y 552.142,Z 404.71,A -85,B 0,C 180,E1 -3356.15,E2 -3356.15} C_VEL
LIN {X 0,Y 552.056,Z 404.717,A -85,B 0,C 180,E1 -3358.932,E2 -3358.932} C_VEL
LIN {X 0,Y 552.114,Z 404.716,A -85,B 0,C 180,E1 -3361.476,E2 -3361.476} C_VEL
LIN {X 0,Y 552.132,Z 404.707,A -85,B 0,C 180,E1 -3364.17,E2 -3364.17} C_VEL
LIN {X 0,Y 552.1,Z 404.71,A -85,B 0,C 180,E1 -3366.748,E2 -3366.748} C_VEL
LIN {X 0,Y 552.13,Z 404.713,A -85,B 0,C 180,E1 -3369.527,E2 -3369.527} C_VEL
LIN {X 0,Y 552.112,Z 404.707,A -85,B 0,C 180,E1 -3372.427,E2 -3372.427} C_VEL
LIN {X 0,Y 552.099,Z 404.713,A -85,B 0,C 180,E1 -3375.563,E2 -3375.563} C_VEL
LIN {X 0,Y 552.124,Z 404.707,A -85,B 0,C 180,E1 -3378.554,E2 -3378.554} C_VEL
LIN {X 0,Y 552.121,Z 404.711,A -85,B 0,C 180,E1 -3381.411,E2 -3381.411} C_VEL
LIN {X 0,Y 552.089,Z 404.71,A -85,B 0,C 180,E1 -3384.156,E2 -3384.156} C_VEL
LIN {X 0,Y 552.118,Z 404.713,A -85,B 0,C 180,E1 -3386.814,E2 -3386.814} C_VEL
LIN {X 0,Y 552.105,Z 404.711,A -85,B 0,C 180,E1 -3389.391,E2 -3389.391} C_VEL
LIN {X 0,Y 552.099,Z 404.709,A -85,B 0,C 180,E1 -3391.901,E2 -3391.901} C_VEL
LIN {X 0,Y 552.14,Z 404.712,A -85,B 0,C 180,E1 -3394.654,E2 -3394.654} C_VEL
LIN {X 0,Y 552.095,Z 404.711,A -85,B 0,C 180,E1 -3397.549,E2 -3397.549} C_VEL
LIN {X 0,Y 552.148,Z 404.71,A -85,B 0,C 180,E1 -3400.375,E2 -3400.375} C_VEL
LIN {X 0,Y 552.121,Z 404.711,A -85,B 0,C 180,E1 -3402.976,E2 -3402.976} C_VEL
LIN {X 0,Y 552.128,Z 404.71,A -85,B 0,C 180,E1 -3405.732,E2 -3405.732} C_VEL
LIN {X 0,Y 553.416,Z 410.933,A -85,B 0,C 180,E1 -3405.849,E2 -3405.849} C_VEL
LIN {X 0,Y 553.13,Z 507.669,A -85,B 0,C 180,E1 -3407.129,E2 -3407.129} C_VEL
LIN {X 0,Y 553.008,Z 520.584,A -85,B 0,C 180,E1 -3407.43,E2 -3407.43} C_VEL
LIN {X 0,Y 552.835,Z 533.318,A -85,B 0,C 180,E1 -3407.892,E2 -3407.892} C_VEL
LIN {X 0,Y 552.684,Z 543.867,A -85,B 0,C 180,E1 -3408.402,E2 -3408.402} C_VEL
LIN {X 0,Y 552.604,Z 552.667,A -85,B 0,C 180,E1 -3408.927,E2 -3408.927} C_VEL
LIN {X 0,Y 552.436,Z 561.445,A -85,B 0,C 180,E1 -3409.555,E2 -3409.555} C_VEL
LIN {X 0,Y 552.245,Z 570.058,A -85,B 0,C 180,E1 -3410.292,E2 -3410.292} C_VEL
LIN {X 0,Y 552.083,Z 579.009,A -85,B 0,C 180,E1 -3411.213,E2 -3411.213} C_VEL
LIN {X 0,Y 551.95,Z 587.671,A -85,B 0,C 180,E1 -3412.317,E2 -3412.317} C_VEL
LIN {X 0,Y 551.843,Z 594.567,A -85,B 0,C 180,E1 -3413.418,E2 -3413.418} C_VEL
LIN {X 0,Y 551.868,Z 598.453,A -85,B 0,C 180,E1 -3414.153,E2 -3414.153} C_VEL
LIN {X 0,Y 551.725,Z 603.164,A -85,B 0,C 180,E1 -3415.251,E2 -3415.251} C_VEL
LIN {X 0,Y 551.75,Z 606.788,A -85,B 0,C 180,E1 -3416.348,E2 -3416.348} C_VEL
LIN {X 0,Y 551.723,Z 608.691,A -85,B 0,C 180,E1 -3417.079,E2 -3417.079} C_VEL
LIN {X 0,Y 551.656,Z 610.126,A -85,B 0,C 180,E1 -3417.81,E2 -3417.81} C_VEL
LIN {X 0,Y 551.642,Z 611.739,A -85,B 0,C 180,E1 -3419.27,E2 -3419.27} C_VEL
LIN {X 0,Y 551.641,Z 611.996,A -85,B 0,C 180,E1 -3420,E2 -3420} C_VEL
LIN {X 0,Y 551.645,Z 611.202,A -85,B 0,C 180,E1 -3421.46,E2 -3421.46} C_VEL
LIN {X 0,Y 551.657,Z 610.283,A -85,B 0,C 180,E1 -3422.19,E2 -3422.19} C_VEL
LIN {X 0,Y 551.724,Z 608.864,A -85,B 0,C 180,E1 -3422.921,E2 -3422.921} C_VEL
LIN {X 0,Y 551.764,Z 604.829,A -85,B 0,C 180,E1 -3424.383,E2 -3424.383} C_VEL
LIN {X 0,Y 551.803,Z 600.536,A -85,B 0,C 180,E1 -3425.481,E2 -3425.481} C_VEL
LIN {X 0,Y 551.824,Z 595.064,A -85,B 0,C 180,E1 -3426.582,E2 -3426.582} C_VEL
LIN {X 0,Y 551.925,Z 589.483,A -85,B 0,C 180,E1 -3427.5,E2 -3427.5} C_VEL
LIN {X 0,Y 552.025,Z 582.789,A -85,B 0,C 180,E1 -3428.419,E2 -3428.419} C_VEL
LIN {X 0,Y 552.165,Z 574.753,A -85,B 0,C 180,E1 -3429.34,E2 -3429.34} C_VEL
LIN {X 0,Y 552.395,Z 563.763,A -85,B 0,C 180,E1 -3430.353,E2 -3430.353} C_VEL
LIN {X 0,Y 552.528,Z 554.015,A -85,B 0,C 180,E1 -3431.075,E2 -3431.075} C_VEL
LIN {X 0,Y 552.702,Z 544.209,A -85,B 0,C 180,E1 -3431.669,E2 -3431.669} C_VEL
LIN {X 0,Y 552.784,Z 534.275,A -85,B 0,C 180,E1 -3432.156,E2 -3432.156} C_VEL
LIN {X 0,Y 553.018,Z 521.974,A -85,B 0,C 180,E1 -3432.617,E2 -3432.617} C_VEL
LIN {X 0,Y 553.115,Z 508.837,A -85,B 0,C 180,E1 -3432.941,E2 -3432.941} C_VEL
LIN {X 0,Y 553.27,Z 478.704,A -85,B 0,C 180,E1 -3433.358,E2 -3433.358} C_VEL
LIN {X 0,Y 553.328,Z 409.908,A -85,B 0,C 180,E1 -3434.257,E2 -3434.257} C_VEL
LIN {X 0,Y 552.126,Z 404.709,A -85,B 0,C 180,E1 -3434.379,E2 -3434.379} C_VEL
LIN {X 0,Y 552.1,Z 404.715,A -85,B 0,C 180,E1 -3437.307,E2 -3437.307} C_VEL
LIN {X 0,Y 552.125,Z 404.708,A -85,B 0,C 180,E1 -3440.14,E2 -3440.14} C_VEL
LIN {X 0,Y 551.426,Z 404.795,A -85,B 0,C 180,E1 -3440.749,E2 -3440.749} C_VEL
LIN {X 0,Y 548.533,Z 405.157,A -85,B 0,C 180,E1 -3441.736,E2 -3441.736} C_VEL
LIN {X 0,Y 546.125,Z 405.454,A -85,B 0,C 180,E1 -3442.531,E2 -3442.531} C_VEL
LIN {X 0,Y 545.123,Z 405.582,A -85,B 0,C 180,E1 -3443.145,E2 -3443.145} C_VEL
LIN {X 0,Y 545.058,Z 405.589,A -85,B 0,C 180,E1 -3443.353,E2 -3443.353} C_VEL
LIN {X 0,Y 545.065,Z 405.585,A -85,B 0,C 180,E1 -3446.001,E2 -3446.001} C_VEL
LIN {X 0,Y 545.078,Z 405.584,A -85,B 0,C 180,E1 -3448.745,E2 -3448.745} C_VEL
LIN {X 0,Y 545.061,Z 405.585,A -85,B 0,C 180,E1 -3451.679,E2 -3451.679} C_VEL
LIN {X 0,Y 545.065,Z 405.582,A -85,B 0,C 180,E1 -3454.564,E2 -3454.564} C_VEL
LIN {X 0,Y 545.04,Z 405.593,A -85,B 0,C 180,E1 -3457.304,E2 -3457.304} C_VEL
LIN {X 0,Y 545.069,Z 405.581,A -85,B 0,C 180,E1 -3460.143,E2 -3460.143} C_VEL
LIN {X 0,Y 545.082,Z 405.589,A -85,B 0,C 180,E1 -3463.107,E2 -3463.107} C_VEL
LIN {X 0,Y 545.06,Z 405.584,A -85,B 0,C 180,E1 -3466.225,E2 -3466.225} C_VEL
LIN {X 0,Y 545.084,Z 405.587,A -85,B 0,C 180,E1 -3468.885,E2 -3468.885} C_VEL
LIN {X 0,Y 545.082,Z 405.59,A -85,B 0,C 180,E1 -3470.818,E2 -3470.818} C_VEL
LIN {X 0,Y 545.037,Z 405.587,A -85,B 0,C 180,E1 -3473.619,E2 -3473.619} C_VEL
LIN {X 0,Y 545.068,Z 405.591,A -85,B 0,C 180,E1 -3476.328,E2 -3476.328} C_VEL
LIN {X 0,Y 545.065,Z 405.588,A -85,B 0,C 180,E1 -3478.952,E2 -3478.952} C_VEL
LIN {X 0,Y 545.046,Z 405.589,A -85,B 0,C 180,E1 -3481.504,E2 -3481.504} C_VEL
LIN {X 0,Y 545.037,Z 405.596,A -85,B 0,C 180,E1 -3484.505,E2 -3484.505} C_VEL
LIN {X 0,Y 545.09,Z 405.686,A -85,B 0,C 180,E1 -3485.995,E2 -3485.995} C_VEL
LIN {X 0,Y 546.264,Z 412.808,A -85,B 0,C 180,E1 -3487.096,E2 -3487.096} C_VEL
LIN {X 0,Y 545.981,Z 432.501,A -85,B 0,C 180,E1 -3489.998,E2 -3489.998} C_VEL
LIN {X 0,Y 545.657,Z 451.313,A -85,B 0,C 180,E1 -3492.768,E2 -3492.768} C_VEL
LIN {X 0,Y 545.398,Z 469.682,A -85,B 0,C 180,E1 -3495.478,E2 -3495.478} C_VEL
LIN {X 0,Y 546.489,Z 478.12,A -85,B 0,C 180,E1 -3495.628,E2 -3495.628} C_VEL
LIN {X 0,Y 546.206,Z 576.283,A -85,B 0,C 180,E1 -3496.94,E2 -3496.94} C_VEL
LIN {X 0,Y 546.105,Z 586.138,A -85,B 0,C 180,E1 -3497.15,E2 -3497.15} C_VEL
LIN {X 0,Y 545.996,Z 596.087,A -85,B 0,C 180,E1 -3497.455,E2 -3497.455} C_VEL
LIN {X 0,Y 545.863,Z 605.429,A -85,B 0,C 180,E1 -3497.829,E2 -3497.829} C_VEL
LIN {X 0,Y 545.712,Z 615.631,A -85,B 0,C 180,E1 -3498.35,E2 -3498.35} C_VEL
LIN {X 0,Y 545.536,Z 625.164,A -85,B 0,C 180,E1 -3498.952,E2 -3498.952} C_VEL
LIN {X 0,Y 545.381,Z 633.755,A -85,B 0,C 180,E1 -3499.606,E2 -3499.606} C_VEL
LIN {X 0,Y 545.164,Z 641.985,A -85,B 0,C 180,E1 -3500.352,E2 -3500.352} C_VEL
LIN {X 0,Y 545.068,Z 648.974,A -85,B 0,C 180,E1 -3501.099,E2 -3501.099} C_VEL
LIN {X 0,Y 544.916,Z 656.304,A -85,B 0,C 180,E1 -3502.03,E2 -3502.03} C_VEL
LIN {X 0,Y 544.822,Z 662.418,A -85,B 0,C 180,E1 -3502.961,E2 -3502.961} C_VEL
LIN {X 0,Y 544.77,Z 667.385,A -85,B 0,C 180,E1 -3503.864,E2 -3503.864} C_VEL
LIN {X 0,Y 544.653,Z 671.724,A -85,B 0,C 180,E1 -3504.818,E2 -3504.818} C_VEL
LIN {X 0,Y 544.684,Z 675.703,A -85,B 0,C 180,E1 -3505.931,E2 -3505.931} C_VEL
LIN {X 0,Y 544.65,Z 678.654,A -85,B 0,C 180,E1 -3507.041,E2 -3507.041} C_VEL
LIN {X 0,Y 544.571,Z 680.142,A -85,B 0,C 180,E1 -3507.781,E2 -3507.781} C_VEL
LIN {X 0,Y 544.542,Z 681.724,A -85,B 0,C 180,E1 -3509.261,E2 -3509.261} C_VEL
LIN {X 0,Y 544.542,Z 681.996,A -85,B 0,C 180,E1 -3510,E2 -3510} C_VEL
LIN {X 0,Y 544.546,Z 681.208,A -85,B 0,C 180,E1 -3511.479,E2 -3511.479} C_VEL
LIN {X 0,Y 544.572,Z 680.28,A -85,B 0,C 180,E1 -3512.219,E2 -3512.219} C_VEL
LIN {X 0,Y 544.669,Z 677.046,A -85,B 0,C 180,E1 -3513.699,E2 -3513.699} C_VEL
LIN {X 0,Y 544.628,Z 673.486,A -85,B 0,C 180,E1 -3514.811,E2 -3514.811} C_VEL
LIN {X 0,Y 544.767,Z 668.832,A -85,B 0,C 180,E1 -3515.924,E2 -3515.924} C_VEL
LIN {X 0,Y 544.785,Z 664.03,A -85,B 0,C 180,E1 -3516.853,E2 -3516.853} C_VEL
LIN {X 0,Y 544.895,Z 658.24,A -85,B 0,C 180,E1 -3517.783,E2 -3517.783} C_VEL
LIN {X 0,Y 545.016,Z 651.277,A -85,B 0,C 180,E1 -3518.715,E2 -3518.715} C_VEL
LIN {X 0,Y 545.134,Z 644.716,A -85,B 0,C 180,E1 -3519.461,E2 -3519.461} C_VEL
LIN {X 0,Y 545.285,Z 635.901,A -85,B 0,C 180,E1 -3520.302,E2 -3520.302} C_VEL
LIN {X 0,Y 545.492,Z 627.728,A -85,B 0,C 180,E1 -3520.955,E2 -3520.955} C_VEL
LIN {X 0,Y 545.646,Z 619.256,A -85,B 0,C 180,E1 -3521.526,E2 -3521.526} C_VEL
LIN {X 0,Y 545.788,Z 609.269,A -85,B 0,C 180,E1 -3522.078,E2 -3522.078} C_VEL
LIN {X 0,Y 545.911,Z 599.752,A -85,B 0,C 180,E1 -3522.5,E2 -3522.5} C_VEL
LIN {X 0,Y 546.104,Z 589.414,A -85,B 0,C 180,E1 -3522.85,E2 -3522.85} C_VEL
LIN {X 0,Y 546.191,Z 578.668,A -85,B 0,C 180,E1 -3523.108,E2 -3523.108} C_VEL
LIN {X 0,Y 546.357,Z 552.238,A -85,B 0,C 180,E1 -3523.483,E2 -3523.483} C_VEL
LIN {X 0,Y 546.419,Z 476.526,A -85,B 0,C 180,E1 -3524.485,E2 -3524.485} C_VEL
LIN {X 0,Y 545.394,Z 469.579,A -85,B 0,C 180,E1 -3524.627,E2 -3524.627} C_VEL
LIN {X 0,Y 545.701,Z 448.385,A -85,B 0,C 180,E1 -3527.754,E2 -3527.754} C_VEL
LIN {X 0,Y 546.037,Z 428.201,A -85,B 0,C 180,E1 -3530.729,E2 -3530.729} C_VEL
LIN {X 0,Y 546.209,Z 412.114,A -85,B 0,C 180,E1 -3533.106,E2 -3533.106} C_VEL
LIN {X 0,Y 545.067,Z 405.593,A -85,B 0,C 180,E1 -3534.122,E2 -3534.122} C_VEL
LIN {X 0,Y 545.029,Z 405.594,A -85,B 0,C 180,E1 -3537.159,E2 -3537.159} C_VEL
LIN {X 0,Y 545.064,Z 405.588,A -85,B 0,C 180,E1 -3540.19,E2 -3540.19} C_VEL
LIN {X 0,Y 545.082,Z 405.587,A -85,B 0,C 180,E1 -3543.062,E2 -3543.062} C_VEL
LIN {X 0,Y 545.028,Z 405.596,A -85,B 0,C 180,E1 -3545.672,E2 -3545.672} C_VEL
LIN {X 0,Y 545.052,Z 405.587,A -85,B 0,C 180,E1 -3548.238,E2 -3548.238} C_VEL
LIN {X 0,Y 545.084,Z 405.582,A -85,B 0,C 180,E1 -3550.473,E2 -3550.473} C_VEL
LIN {X 0,Y 545.082,Z 405.59,A -85,B 0,C 180,E1 -3553.107,E2 -3553.107} C_VEL
LIN {X 0,Y 545.071,Z 405.585,A -85,B 0,C 180,E1 -3556.224,E2 -3556.224} C_VEL
LIN {X 0,Y 545.085,Z 405.588,A -85,B 0,C 180,E1 -3558.885,E2 -3558.885} C_VEL
LIN {X 0,Y 545.086,Z 405.592,A -85,B 0,C 180,E1 -3560.819,E2 -3560.819} C_VEL
LIN {X 0,Y 545.037,Z 405.584,A -85,B 0,C 180,E1 -3563.619,E2 -3563.619} C_VEL
LIN {X 0,Y 545.068,Z 405.589,A -85,B 0,C 180,E1 -3566.328,E2 -3566.328} C_VEL
LIN {X 0,Y 545.065,Z 405.588,A -85,B 0,C 180,E1 -3568.952,E2 -3568.952} C_VEL
LIN {X 0,Y 545.047,Z 405.588,A -85,B 0,C 180,E1 -3571.504,E2 -3571.504} C_VEL
LIN {X 0,Y 545.039,Z 405.596,A -85,B 0,C 180,E1 -3574.504,E2 -3574.504} C_VEL
LIN {X 0,Y 545.074,Z 405.715,A -85,B 0,C 180,E1 -3575.968,E2 -3575.968} C_VEL
LIN {X 0,Y 546.307,Z 413.088,A -85,B 0,C 180,E1 -3577.098,E2 -3577.098} C_VEL
LIN {X 0,Y 545.972,Z 433.225,A -85,B 0,C 180,E1 -3580.111,E2 -3580.111} C_VEL
LIN {X 0,Y 545.626,Z 452.562,A -85,B 0,C 180,E1 -3582.96,E2 -3582.96} C_VEL
LIN {X 0,Y 545.397,Z 469.707,A -85,B 0,C 180,E1 -3585.482,E2 -3585.482} C_VEL
LIN {X 0,Y 546.496,Z 478.29,A -85,B 0,C 180,E1 -3585.63,E2 -3585.63} C_VEL
LIN {X 0,Y 546.206,Z 576.319,A -85,B 0,C 180,E1 -3586.94,E2 -3586.94} C_VEL
LIN {X 0,Y 546.081,Z 587.022,A -85,B 0,C 180,E1 -3587.173,E2 -3587.173} C_VEL
LIN {X 0,Y 545.968,Z 597.373,A -85,B 0,C 180,E1 -3587.501,E2 -3587.501} C_VEL
LIN {X 0,Y 545.826,Z 608.453,A -85,B 0,C 180,E1 -3587.97,E2 -3587.97} C_VEL
LIN {X 0,Y 545.641,Z 620.875,A -85,B 0,C 180,E1 -3588.66,E2 -3588.66} C_VEL
LIN {X 0,Y 545.402,Z 631.457,A -85,B 0,C 180,E1 -3589.419,E2 -3589.419} C_VEL
LIN {X 0,Y 545.222,Z 640.054,A -85,B 0,C 180,E1 -3590.166,E2 -3590.166} C_VEL
LIN {X 0,Y 545.101,Z 647.309,A -85,B 0,C 180,E1 -3590.913,E2 -3590.913} C_VEL
LIN {X 0,Y 544.922,Z 654.934,A -85,B 0,C 180,E1 -3591.844,E2 -3591.844} C_VEL
LIN {X 0,Y 544.827,Z 661.279,A -85,B 0,C 180,E1 -3592.775,E2 -3592.775} C_VEL
LIN {X 0,Y 544.761,Z 667.424,A -85,B 0,C 180,E1 -3593.871,E2 -3593.871} C_VEL
LIN {X 0,Y 544.64,Z 673.22,A -85,B 0,C 180,E1 -3595.189,E2 -3595.189} C_VEL
LIN {X 0,Y 544.669,Z 676.848,A -85,B 0,C 180,E1 -3596.301,E2 -3596.301} C_VEL
LIN {X 0,Y 544.65,Z 678.67,A -85,B 0,C 180,E1 -3597.041,E2 -3597.041} C_VEL
LIN {X 0,Y 544.546,Z 681.147,A -85,B 0,C 180,E1 -3598.521,E2 -3598.521} C_VEL
LIN {X 0,Y 544.542,Z 681.748,A -85,B 0,C 180,E1 -3599.26,E2 -3599.26} C_VEL
LIN {X 0,Y 544.542,Z 681.808,A -85,B 0,C 180,E1 -3600.739,E2 -3600.739} C_VEL
LIN {X 0,Y 544.546,Z 681.228,A -85,B 0,C 180,E1 -3601.479,E2 -3601.479} C_VEL
LIN {X 0,Y 544.651,Z 678.883,A -85,B 0,C 180,E1 -3602.959,E2 -3602.959} C_VEL
LIN {X 0,Y 544.684,Z 676,A -85,B 0,C 180,E1 -3604.069,E2 -3604.069} C_VEL
LIN {X 0,Y 544.653,Z 672.083,A -85,B 0,C 180,E1 -3605.182,E2 -3605.182} C_VEL
LIN {X 0,Y 544.762,Z 667.89,A -85,B 0,C 180,E1 -3606.129,E2 -3606.129} C_VEL
LIN {X 0,Y 544.822,Z 661.842,A -85,B 0,C 180,E1 -3607.225,E2 -3607.225} C_VEL
LIN {X 0,Y 544.915,Z 655.606,A -85,B 0,C 180,E1 -3608.156,E2 -3608.156} C_VEL
LIN {X 0,Y 545.026,Z 649.758,A -85,B 0,C 180,E1 -3608.902,E2 -3608.902} C_VEL
LIN {X 0,Y 545.159,Z 642.941,A -85,B 0,C 180,E1 -3609.648,E2 -3609.648} C_VEL
LIN {X 0,Y 545.387,Z 633.714,A -85,B 0,C 180,E1 -3610.487,E2 -3610.487} C_VEL
LIN {X 0,Y 545.526,Z 625.112,A -85,B 0,C 180,E1 -3611.142,E2 -3611.142} C_VEL
LIN {X 0,Y 545.721,Z 615.131,A -85,B 0,C 180,E1 -3611.768,E2 -3611.768} C_VEL
LIN {X 0,Y 545.835,Z 604.285,A -85,B 0,C 180,E1 -3612.313,E2 -3612.313} C_VEL
LIN {X 0,Y 546.07,Z 591.226,A -85,B 0,C 180,E1 -3612.804,E2 -3612.804} C_VEL
LIN {X 0,Y 546.189,Z 578.734,A -85,B 0,C 180,E1 -3613.108,E2 -3613.108} C_VEL
LIN {X 0,Y 546.338,Z 550.453,A -85,B 0,C 180,E1 -3613.507,E2 -3613.507} C_VEL
LIN {X 0,Y 546.414,Z 476.271,A -85,B 0,C 180,E1 -3614.489,E2 -3614.489} C_VEL
LIN {X 0,Y 545.392,Z 469.69,A -85,B 0,C 180,E1 -3614.611,E2 -3614.611} C_VEL
LIN {X 0,Y 545.672,Z 449.234,A -85,B 0,C 180,E1 -3617.619,E2 -3617.619} C_VEL
LIN {X 0,Y 546.039,Z 430.818,A -85,B 0,C 180,E1 -3620.335,E2 -3620.335} C_VEL
LIN {X 0,Y 546.138,Z 412.698,A -85,B 0,C 180,E1 -3622.909,E2 -3622.909} C_VEL
LIN {X 0,Y 545.068,Z 405.593,A -85,B 0,C 180,E1 -3623.984,E2 -3623.984} C_VEL
LIN {X 0,Y 545.029,Z 405.594,A -85,B 0,C 180,E1 -3627.159,E2 -3627.159} C_VEL
LIN {X 0,Y 545.064,Z 405.589,A -85,B 0,C 180,E1 -3630.19,E2 -3630.19} C_VEL
LIN {X 0,Y 545.082,Z 405.587,A -85,B 0,C 180,E1 -3633.062,E2 -3633.062} C_VEL
LIN {X 0,Y 545.028,Z 405.595,A -85,B 0,C 180,E1 -3635.672,E2 -3635.672} C_VEL
LIN {X 0,Y 545.052,Z 405.587,A -85,B 0,C 180,E1 -3638.237,E2 -3638.237} C_VEL
LIN {X 0,Y 545.083,Z 405.584,A -85,B 0,C 180,E1 -3640.473,E2 -3640.473} C_VEL
LIN {X 0,Y 545.081,Z 405.59,A -85,B 0,C 180,E1 -3643.107,E2 -3643.107} C_VEL
LIN {X 0,Y 545.07,Z 405.586,A -85,B 0,C 180,E1 -3646.224,E2 -3646.224} C_VEL
LIN {X 0,Y 545.084,Z 405.59,A -85,B 0,C 180,E1 -3648.885,E2 -3648.885} C_VEL
LIN {X 0,Y 545.082,Z 405.59,A -85,B 0,C 180,E1 -3650.818,E2 -3650.818} C_VEL
LIN {X 0,Y 545.037,Z 405.589,A -85,B 0,C 180,E1 -3653.619,E2 -3653.619} C_VEL
LIN {X 0,Y 545.068,Z 405.59,A -85,B 0,C 180,E1 -3656.328,E2 -3656.328} C_VEL
LIN {X 0,Y 545.065,Z 405.589,A -85,B 0,C 180,E1 -3658.952,E2 -3658.952} C_VEL
LIN {X 0,Y 545.045,Z 405.59,A -85,B 0,C 180,E1 -3661.504,E2 -3661.504} C_VEL
LIN {X 0,Y 545.068,Z 405.604,A -85,B 0,C 180,E1 -3663.51,E2 -3663.51} C_VEL
LIN {X 0,Y 546.857,Z 414.345,A -85,B 0,C 180,E1 -3664.737,E2 -3664.737} C_VEL
LIN {X 0,Y 546.492,Z 436.703,A -85,B 0,C 180,E1 -3667.624,E2 -3667.624} C_VEL
LIN {X 0,Y 546.135,Z 458.022,A -85,B 0,C 180,E1 -3670.324,E2 -3670.324} C_VEL
LIN {X 0,Y 545.788,Z 480.657,A -85,B 0,C 180,E1 -3673.158,E2 -3673.158} C_VEL
LIN {X 0,Y 545.508,Z 498.668,A -85,B 0,C 180,E1 -3675.43,E2 -3675.43} C_VEL
LIN {X 0,Y 546.535,Z 506.986,A -85,B 0,C 180,E1 -3675.569,E2 -3675.569} C_VEL
LIN {X 0,Y 546.216,Z 607.943,A -85,B 0,C 180,E1 -3676.916,E2 -3676.916} C_VEL
LIN {X 0,Y 546.053,Z 621.215,A -85,B 0,C 180,E1 -3677.243,E2 -3677.243} C_VEL
LIN {X 0,Y 545.883,Z 633.368,A -85,B 0,C 180,E1 -3677.688,E2 -3677.688} C_VEL
LIN {X 0,Y 545.698,Z 645.711,A -85,B 0,C 180,E1 -3678.302,E2 -3678.302} C_VEL
LIN {X 0,Y 545.491,Z 657.194,A -85,B 0,C 180,E1 -3679.045,E2 -3679.045} C_VEL
LIN {X 0,Y 545.29,Z 667.605,A -85,B 0,C 180,E1 -3679.886,E2 -3679.886} C_VEL
LIN {X 0,Y 545.085,Z 676.113,A -85,B 0,C 180,E1 -3680.725,E2 -3680.725} C_VEL
LIN {X 0,Y 544.978,Z 683.96,A -85,B 0,C 180,E1 -3681.658,E2 -3681.658} C_VEL
LIN {X 0,Y 544.824,Z 691.622,A -85,B 0,C 180,E1 -3682.775,E2 -3682.775} C_VEL
LIN {X 0,Y 544.776,Z 698.679,A -85,B 0,C 180,E1 -3684.076,E2 -3684.076} C_VEL
LIN {X 0,Y 544.628,Z 703.373,A -85,B 0,C 180,E1 -3685.189,E2 -3685.189} C_VEL
LIN {X 0,Y 544.669,Z 706.958,A -85,B 0,C 180,E1 -3686.301,E2 -3686.301} C_VEL
LIN {X 0,Y 544.65,Z 708.807,A -85,B 0,C 180,E1 -3687.041,E2 -3687.041} C_VEL
LIN {X 0,Y 544.546,Z 711.183,A -85,B 0,C 180,E1 -3688.521,E2 -3688.521} C_VEL
LIN {X 0,Y 544.541,Z 712,A -85,B 0,C 180,E1 -3690,E2 -3690} C_VEL
LIN {X 0,Y 544.546,Z 711.184,A -85,B 0,C 180,E1 -3691.479,E2 -3691.479} C_VEL
LIN {X 0,Y 544.65,Z 708.81,A -85,B 0,C 180,E1 -3692.959,E2 -3692.959} C_VEL
LIN {X 0,Y 544.684,Z 705.895,A -85,B 0,C 180,E1 -3694.069,E2 -3694.069} C_VEL
LIN {X 0,Y 544.653,Z 701.948,A -85,B 0,C 180,E1 -3695.182,E2 -3695.182} C_VEL
LIN {X 0,Y 544.74,Z 696.703,A -85,B 0,C 180,E1 -3696.328,E2 -3696.328} C_VEL
LIN {X 0,Y 544.836,Z 690.467,A -85,B 0,C 180,E1 -3697.411,E2 -3697.411} C_VEL
LIN {X 0,Y 545.007,Z 682.477,A -85,B 0,C 180,E1 -3698.528,E2 -3698.528} C_VEL
LIN {X 0,Y 545.154,Z 674.333,A -85,B 0,C 180,E1 -3699.461,E2 -3699.461} C_VEL
LIN {X 0,Y 545.369,Z 664.397,A -85,B 0,C 180,E1 -3700.394,E2 -3700.394} C_VEL
LIN {X 0,Y 545.548,Z 654.59,A -85,B 0,C 180,E1 -3701.142,E2 -3701.142} C_VEL
LIN {X 0,Y 545.694,Z 643.578,A -85,B 0,C 180,E1 -3701.817,E2 -3701.817} C_VEL
LIN {X 0,Y 545.896,Z 631.101,A -85,B 0,C 180,E1 -3702.406,E2 -3702.406} C_VEL
LIN {X 0,Y 546.095,Z 618.084,A -85,B 0,C 180,E1 -3702.85,E2 -3702.85} C_VEL
LIN {X 0,Y 546.22,Z 605.099,A -85,B 0,C 180,E1 -3703.131,E2 -3703.131} C_VEL
LIN {X 0,Y 546.451,Z 505.372,A -85,B 0,C 180,E1 -3704.455,E2 -3704.455} C_VEL
LIN {X 0,Y 545.514,Z 498.5,A -85,B 0,C 180,E1 -3704.592,E2 -3704.592} C_VEL
LIN {X 0,Y 545.858,Z 475.633,A -85,B 0,C 180,E1 -3707.456,E2 -3707.456} C_VEL
LIN {X 0,Y 546.217,Z 450.754,A -85,B 0,C 180,E1 -3710.525,E2 -3710.525} C_VEL
LIN {X 0,Y 546.446,Z 426.988,A -85,B 0,C 180,E1 -3713.497,E2 -3713.497} C_VEL
LIN {X 0,Y 546.533,Z 412.967,A -85,B 0,C 180,E1 -3715.269,E2 -3715.269} C_VEL
LIN {X 0,Y 545.071,Z 405.59,A -85,B 0,C 180,E1 -3716.284,E2 -3716.284} C_VEL
LIN {X 0,Y 545.031,Z 405.596,A -85,B 0,C 180,E1 -3719.341,E2 -3719.341} C_VEL
